(* Logix 5000 project; controller reports 1756-L63 rev 20.11; software revision 20.04; part 33 of 52 *)

        [12].log_data[39].valid := 1, [12].log_data[40].min := 7.5629425, [12].log_data[40].max := 7.590698, [12].log_data[40].total := 27279.617, [12].log_data[40].time := 3600.0, [12].log_data[40].minminute := 8, [12].log_data[40].maxminute := 16, [12].log_data[40].valid := 1, [12].log_data[41].min := 0.03412134, [12].log_data[41].max := 0.0517876, [12].log_data[41].total := 150.64825, [12].log_data[41].time := 3600.0, [12].log_data[41].minminute := 1, [12].log_data[41].maxminute := 24, [12].log_data[41].valid := 1, [12].log_data[42].min := 2.292585, [12].log_data[42].max := 2.2987092, [12].log_data[42].total := 8264.11, [12].log_data[42].time := 3600.0, [12].log_data[42].minminute := 1, [12].log_data[42].maxminute := 32, [12].log_data[42].valid := 1, [12].log_data[43].min := -0.27999878, [12].log_data[43].max := -0.26000214, [12].log_data[43].total := -938.01764, [12].log_data[43].time := 3600.0, [12].log_data[43].valid := 1, [12].log_data[44].min := -0.30000305, [12].log_data[44].max := -0.27999878, [12].log_data[44].total := -1080.081, [12].log_data[44].time := 3600.0, [12].log_data[44].maxminute := 16, [12].log_data[44].valid := 1, [12].log_data[45].time := 3600.0, [12].log_data[45].valid := 1, [12].log_data[46].time := 3600.0, [12].log_data[46].valid := 1, [12].log_data[47].time := 3600.0, [12].log_data[47].valid := 1, [12].log_data[48].min := 6.650855, [12].log_data[48].max := 6.8709764, [12].log_data[48].total := 24089.69, [12].log_data[48].time := 3600.0, [12].log_data[48].minminute := 16, [12].log_data[48].maxminute := 3, [12].log_data[48].valid := 1, [12].log_data[49].min := 7.641001, [12].log_data[49].max := 9.442957, [12].log_data[49].total := 31503.416, [12].log_data[49].time := 3600.0, [12].log_data[49].minminute := 15, [12].log_data[49].maxminute := 59, [12].log_data[49].valid := 1, [12].log_data[50].min := 2.016285, [12].log_data[50].max := 2.093074, [12].log_data[50].total := 7406.019, [12].log_data[50].time := 3600.0, [12].log_data[50].minminute := 59, [12].log_data[50].maxminute := 5, [12].log_data[50].valid := 1,
        [12].log_data[51].time := 3600.0, [12].log_data[51].valid := 1, [12].log_data[52].min := -2.9199982, [12].log_data[52].max := 0.11999512, [12].log_data[52].total := -7511.6816, [12].log_data[52].time := 3600.0, [12].log_data[52].minminute := 12, [12].log_data[52].valid := 1, [12].log_data[53].min := -2.5, [12].log_data[53].max := 0.19999695, [12].log_data[53].total := -7003.9526, [12].log_data[53].time := 3600.0, [12].log_data[53].minminute := 37, [12].log_data[53].maxminute := 15, [12].log_data[53].valid := 1, [12].log_data[54].max := 0.535, [12].log_data[54].total := 1217.1705, [12].log_data[54].time := 3600.0, [12].log_data[54].maxminute := 12, [12].log_data[54].valid := 1, [12].log_data[55].max := 0.51600003, [12].log_data[55].total := 1217.1682, [12].log_data[55].time := 3600.0, [12].log_data[55].minminute := 3, [12].log_data[55].maxminute := 37, [12].log_data[55].valid := 1, [12].log_data[56].min := 0.16024561, [12].log_data[56].max := 0.16063818, [12].log_data[56].total := 577.4149, [12].log_data[56].time := 3600.0, [12].log_data[56].minminute := 10, [12].log_data[56].maxminute := 2, [12].log_data[56].valid := 1, [12].log_data[57].min := 0.31213588, [12].log_data[57].max := 0.3125677, [12].log_data[57].total := 1124.3689, [12].log_data[57].time := 3600.0, [12].log_data[57].minminute := 57, [12].log_data[57].maxminute := 15, [12].log_data[57].valid := 1, [12].log_data[58].time := 3600.0, [12].log_data[58].valid := 1, [12].log_data[59].time := 3600.0, [12].log_data[59].valid := 1, [12].log_data[60].valid := 1, [12].log_data[61].valid := 1, [12].log_data[62].valid := 1, [12].log_data[63].valid := 1, [12].log_data[64].valid := 1, [12].log_data[65].valid := 1, [12].log_data[66].valid := 1, [12].log_data[67].valid := 1, [12].log_data[68].valid := 1, [12].log_data[69].valid := 1, [12].log_data[70].valid := 1, [12].log_data[71].valid := 1, [12].log_data[72].valid := 1, [12].log_data[73].valid := 1, [12].log_data[74].valid := 1, [12].log_data[75].valid := 1,
        [12].log_data[76].valid := 1, [12].log_data[77].valid := 1, [12].log_data[78].valid := 1, [12].log_data[79].valid := 1, [12].log_data[80].valid := 1, [12].log_data[81].valid := 1, [12].log_data[82].valid := 1, [12].log_data[83].valid := 1, [12].log_data[84].valid := 1, [12].log_data[85].valid := 1, [12].log_data[86].valid := 1, [12].log_data[87].valid := 1, [12].log_data[88].valid := 1, [12].log_data[89].valid := 1, [12].log_data[90].valid := 1, [12].log_data[91].valid := 1, [12].log_data[92].valid := 1, [12].log_data[93].valid := 1, [12].log_data[94].valid := 1, [12].log_data[95].valid := 1, [12].log_data[96].valid := 1, [12].log_data[97].valid := 1, [12].log_data[98].valid := 1, [12].log_data[99].valid := 1, [12].log_data[100].valid := 1, [12].log_data[101].valid := 1, [12].log_data[102].valid := 1, [12].log_data[103].valid := 1, [12].log_data[104].valid := 1, [12].log_data[105].valid := 1, [12].log_data[106].valid := 1, [12].log_data[107].valid := 1, [12].log_data[108].valid := 1, [12].log_data[109].valid := 1, [12].log_data[110].valid := 1, [12].log_data[111].valid := 1, [12].log_data[112].valid := 1, [12].log_data[113].valid := 1, [12].log_data[114].valid := 1, [12].log_data[115].valid := 1, [12].log_data[116].valid := 1, [12].log_data[117].valid := 1, [12].log_data[118].valid := 1, [12].log_data[119].valid := 1, [12].log_data[120].valid := 1, [12].log_data[121].valid := 1, [12].log_data[122].valid := 1, [12].log_data[123].valid := 1, [12].log_data[124].valid := 1, [12].time.Year := 2023, [12].time.Month := 1, [12].time.Day := 13, [12].time.Hour := 15, [12].time.Minute := 59, [12].time.Second := 59, [13].log_data[0].min := 1.0, [13].log_data[0].max := 1.0, [13].log_data[0].total := 3600.0, [13].log_data[0].time := 3600.0, [13].log_data[0].valid := 1,
        [13].log_data[1].max := 1.0, [13].log_data[1].total := 530.0, [13].log_data[1].time := 3600.0, [13].log_data[1].maxminute := 20, [13].log_data[1].valid := 1, [13].log_data[2].max := 1.0, [13].log_data[2].total := 526.5, [13].log_data[2].time := 3600.0, [13].log_data[2].maxminute := 20, [13].log_data[2].valid := 1, [13].log_data[3].time := 3600.0, [13].log_data[3].valid := 1, [13].log_data[4].time := 3600.0, [13].log_data[4].valid := 1, [13].log_data[5].max := 1.0, [13].log_data[5].total := 238.5, [13].log_data[5].time := 3600.0, [13].log_data[5].maxminute := 23, [13].log_data[5].valid := 1, [13].log_data[6].time := 3600.0, [13].log_data[6].valid := 1, [13].log_data[7].time := 3600.0, [13].log_data[7].valid := 1, [13].log_data[8].max := 1.0, [13].log_data[8].total := 2819.5, [13].log_data[8].time := 3600.0, [13].log_data[8].minminute := 12, [13].log_data[8].valid := 1, [13].log_data[9].max := 1.0, [13].log_data[9].total := 2816.0, [13].log_data[9].time := 3600.0, [13].log_data[9].minminute := 12, [13].log_data[9].valid := 1, [13].log_data[10].min := 1.0, [13].log_data[10].max := 1.0, [13].log_data[10].total := 3600.0, [13].log_data[10].time := 3600.0, [13].log_data[10].valid := 1, [13].log_data[11].time := 3600.0, [13].log_data[11].valid := 1, [13].log_data[12].min := 1.0, [13].log_data[12].max := 1.0, [13].log_data[12].total := 3600.0, [13].log_data[12].time := 3600.0, [13].log_data[12].valid := 1, [13].log_data[13].min := 1.0, [13].log_data[13].max := 1.0, [13].log_data[13].total := 3600.0, [13].log_data[13].time := 3600.0, [13].log_data[13].valid := 1, [13].log_data[14].time := 3600.0, [13].log_data[14].valid := 1, [13].log_data[15].time := 3600.0, [13].log_data[15].valid := 1, [13].log_data[16].time := 3600.0, [13].log_data[16].valid := 1, [13].log_data[17].min := 1.0, [13].log_data[17].max := 1.0, [13].log_data[17].total := 3600.0, [13].log_data[17].time := 3600.0,
        [13].log_data[17].valid := 1, [13].log_data[18].time := 3600.0, [13].log_data[18].valid := 1, [13].log_data[19].time := 3600.0, [13].log_data[19].valid := 1, [13].log_data[20].time := 3600.0, [13].log_data[20].valid := 1, [13].log_data[21].min := 1.0, [13].log_data[21].max := 1.0, [13].log_data[21].total := 3600.0, [13].log_data[21].time := 3600.0, [13].log_data[21].valid := 1, [13].log_data[22].time := 3600.0, [13].log_data[22].valid := 1, [13].log_data[23].time := 3600.0, [13].log_data[23].valid := 1, [13].log_data[24].time := 3600.0, [13].log_data[24].valid := 1, [13].log_data[25].time := 3600.0, [13].log_data[25].valid := 1, [13].log_data[26].time := 3600.0, [13].log_data[26].valid := 1, [13].log_data[27].time := 3600.0, [13].log_data[27].valid := 1, [13].log_data[28].time := 3600.0, [13].log_data[28].valid := 1, [13].log_data[29].min := 1.0, [13].log_data[29].max := 1.0, [13].log_data[29].total := 3600.0, [13].log_data[29].time := 3600.0, [13].log_data[29].valid := 1, [13].log_data[30].min := 1.0, [13].log_data[30].max := 1.0, [13].log_data[30].total := 3600.0, [13].log_data[30].time := 3600.0, [13].log_data[30].valid := 1, [13].log_data[31].max := 1.0, [13].log_data[31].total := 905.749, [13].log_data[31].time := 3600.0, [13].log_data[31].minminute := 3, [13].log_data[31].valid := 1, [13].log_data[32].max := 1.0, [13].log_data[32].total := 1495.5, [13].log_data[32].time := 3600.0, [13].log_data[32].maxminute := 5, [13].log_data[32].valid := 1, [13].log_data[33].time := 3600.0, [13].log_data[33].valid := 1, [13].log_data[34].time := 3600.0, [13].log_data[34].valid := 1, [13].log_data[35].max := 1.0, [13].log_data[35].total := 1299.749, [13].log_data[35].time := 3600.0, [13].log_data[35].minminute := 7, [13].log_data[35].valid := 1, [13].log_data[36].max := 1.0, [13].log_data[36].total := 1160.247, [13].log_data[36].time := 3600.0, [13].log_data[36].maxminute := 8, [13].log_data[36].valid := 1,
        [13].log_data[37].max := 7.6030836, [13].log_data[37].total := 3481.0479, [13].log_data[37].time := 3600.0, [13].log_data[37].maxminute := 21, [13].log_data[37].valid := 1, [13].log_data[38].time := 3600.0, [13].log_data[38].valid := 1, [13].log_data[39].min := 0.9944707, [13].log_data[39].max := 1.02203, [13].log_data[39].total := 3607.03, [13].log_data[39].time := 3600.0, [13].log_data[39].minminute := 59, [13].log_data[39].maxminute := 27, [13].log_data[39].valid := 1, [13].log_data[40].min := 7.572836, [13].log_data[40].max := 7.5805306, [13].log_data[40].total := 27278.973, [13].log_data[40].time := 3600.0, [13].log_data[40].minminute := 17, [13].log_data[40].maxminute := 49, [13].log_data[40].valid := 1, [13].log_data[41].min := 0.028036376, [13].log_data[41].max := 0.049824707, [13].log_data[41].total := 143.90239, [13].log_data[41].time := 3600.0, [13].log_data[41].minminute := 30, [13].log_data[41].maxminute := 4, [13].log_data[41].valid := 1, [13].log_data[42].min := 2.2929382, [13].log_data[42].max := 2.2984736, [13].log_data[42].total := 8264.059, [13].log_data[42].time := 3600.0, [13].log_data[42].minminute := 7, [13].log_data[42].maxminute := 29, [13].log_data[42].valid := 1, [13].log_data[43].min := -0.27999878, [13].log_data[43].max := -0.26000214, [13].log_data[43].total := -938.47235, [13].log_data[43].time := 3600.0, [13].log_data[43].valid := 1, [13].log_data[44].min := -0.30000305, [13].log_data[44].max := -0.27999878, [13].log_data[44].total := -1080.086, [13].log_data[44].time := 3600.0, [13].log_data[44].maxminute := 46, [13].log_data[44].valid := 1, [13].log_data[45].time := 3600.0, [13].log_data[45].valid := 1, [13].log_data[46].time := 3600.0, [13].log_data[46].valid := 1, [13].log_data[47].time := 3600.0, [13].log_data[47].valid := 1, [13].log_data[48].min := 6.5725355, [13].log_data[48].max := 6.936381, [13].log_data[48].total := 24110.77, [13].log_data[48].time := 3600.0, [13].log_data[48].minminute := 50, [13].log_data[48].maxminute := 29, [13].log_data[48].valid := 1, [13].log_data[49].min := 6.7824225,
        [13].log_data[49].max := 9.446097, [13].log_data[49].total := 29833.777, [13].log_data[49].time := 3600.0, [13].log_data[49].minminute := 48, [13].log_data[49].maxminute := 10, [13].log_data[49].valid := 1, [13].log_data[50].min := 1.9995611, [13].log_data[50].max := 2.1512551, [13].log_data[50].total := 7471.418, [13].log_data[50].time := 3600.0, [13].log_data[50].minminute := 12, [13].log_data[50].maxminute := 25, [13].log_data[50].valid := 1, [13].log_data[51].time := 3600.0, [13].log_data[51].valid := 1, [13].log_data[52].min := -4.220001, [13].log_data[52].max := 0.11999512, [13].log_data[52].total := -6930.1035, [13].log_data[52].time := 3600.0, [13].log_data[52].minminute := 25, [13].log_data[52].maxminute := 3, [13].log_data[52].valid := 1, [13].log_data[53].min := -3.959999, [13].log_data[53].max := 0.19999695, [13].log_data[53].total := -6586.3633, [13].log_data[53].time := 3600.0, [13].log_data[53].minminute := 25, [13].log_data[53].maxminute := 31, [13].log_data[53].valid := 1, [13].log_data[54].max := 0.5435, [13].log_data[54].total := 951.75946, [13].log_data[54].time := 3600.0, [13].log_data[54].minminute := 3, [13].log_data[54].maxminute := 28, [13].log_data[54].valid := 1, [13].log_data[55].max := 0.5385, [13].log_data[55].total := 974.7713, [13].log_data[55].time := 3600.0, [13].log_data[55].minminute := 7, [13].log_data[55].maxminute := 25, [13].log_data[55].valid := 1, [13].log_data[56].min := 0.16020635, [13].log_data[56].max := 0.16059892, [13].log_data[56].total := 577.38025, [13].log_data[56].time := 3600.0, [13].log_data[56].minminute := 53, [13].log_data[56].valid := 1, [13].log_data[57].min := 0.31009445, [13].log_data[57].max := 0.31252846, [13].log_data[57].total := 1123.3262, [13].log_data[57].time := 3600.0, [13].log_data[57].minminute := 59, [13].log_data[57].valid := 1, [13].log_data[58].time := 3600.0, [13].log_data[58].valid := 1, [13].log_data[59].time := 3600.0, [13].log_data[59].valid := 1, [13].log_data[60].valid := 1, [13].log_data[61].valid := 1, [13].log_data[62].valid := 1,
        [13].log_data[63].valid := 1, [13].log_data[64].valid := 1, [13].log_data[65].valid := 1, [13].log_data[66].valid := 1, [13].log_data[67].valid := 1, [13].log_data[68].valid := 1, [13].log_data[69].valid := 1, [13].log_data[70].valid := 1, [13].log_data[71].valid := 1, [13].log_data[72].valid := 1, [13].log_data[73].valid := 1, [13].log_data[74].valid := 1, [13].log_data[75].valid := 1, [13].log_data[76].valid := 1, [13].log_data[77].valid := 1, [13].log_data[78].valid := 1, [13].log_data[79].valid := 1, [13].log_data[80].valid := 1, [13].log_data[81].valid := 1, [13].log_data[82].valid := 1, [13].log_data[83].valid := 1, [13].log_data[84].valid := 1, [13].log_data[85].valid := 1, [13].log_data[86].valid := 1, [13].log_data[87].valid := 1, [13].log_data[88].valid := 1, [13].log_data[89].valid := 1, [13].log_data[90].valid := 1, [13].log_data[91].valid := 1, [13].log_data[92].valid := 1, [13].log_data[93].valid := 1, [13].log_data[94].valid := 1, [13].log_data[95].valid := 1, [13].log_data[96].valid := 1, [13].log_data[97].valid := 1, [13].log_data[98].valid := 1, [13].log_data[99].valid := 1, [13].log_data[100].valid := 1, [13].log_data[101].valid := 1, [13].log_data[102].valid := 1, [13].log_data[103].valid := 1, [13].log_data[104].valid := 1, [13].log_data[105].valid := 1, [13].log_data[106].valid := 1, [13].log_data[107].valid := 1, [13].log_data[108].valid := 1, [13].log_data[109].valid := 1, [13].log_data[110].valid := 1, [13].log_data[111].valid := 1, [13].log_data[112].valid := 1, [13].log_data[113].valid := 1, [13].log_data[114].valid := 1, [13].log_data[115].valid := 1, [13].log_data[116].valid := 1, [13].log_data[117].valid := 1, [13].log_data[118].valid := 1, [13].log_data[119].valid := 1, [13].log_data[120].valid := 1, [13].log_data[121].valid := 1, [13].log_data[122].valid := 1,
        [13].log_data[123].valid := 1, [13].log_data[124].valid := 1, [13].time.Year := 2023, [13].time.Month := 1, [13].time.Day := 13, [13].time.Hour := 16, [13].time.Minute := 59, [13].time.Second := 59, [14].log_data[0].min := 1.0, [14].log_data[0].max := 1.0, [14].log_data[0].total := 3600.0, [14].log_data[0].time := 3600.0, [14].log_data[0].valid := 1, [14].log_data[1].time := 3600.0, [14].log_data[1].valid := 1, [14].log_data[2].time := 3600.0, [14].log_data[2].valid := 1, [14].log_data[3].time := 3600.0, [14].log_data[3].valid := 1, [14].log_data[4].time := 3600.0, [14].log_data[4].valid := 1, [14].log_data[5].time := 3600.0, [14].log_data[5].valid := 1, [14].log_data[6].time := 3600.0, [14].log_data[6].valid := 1, [14].log_data[7].time := 3600.0, [14].log_data[7].valid := 1, [14].log_data[8].max := 1.0, [14].log_data[8].total := 3099.251, [14].log_data[8].time := 3600.0, [14].log_data[8].minminute := 51, [14].log_data[8].valid := 1, [14].log_data[9].max := 1.0, [14].log_data[9].total := 3099.251, [14].log_data[9].time := 3600.0, [14].log_data[9].minminute := 51, [14].log_data[9].valid := 1, [14].log_data[10].min := 1.0, [14].log_data[10].max := 1.0, [14].log_data[10].total := 3600.0, [14].log_data[10].time := 3600.0, [14].log_data[10].valid := 1, [14].log_data[11].time := 3600.0, [14].log_data[11].valid := 1, [14].log_data[12].min := 1.0, [14].log_data[12].max := 1.0, [14].log_data[12].total := 3600.0, [14].log_data[12].time := 3600.0, [14].log_data[12].valid := 1, [14].log_data[13].min := 1.0, [14].log_data[13].max := 1.0, [14].log_data[13].total := 3600.0, [14].log_data[13].time := 3600.0, [14].log_data[13].valid := 1, [14].log_data[14].time := 3600.0, [14].log_data[14].valid := 1, [14].log_data[15].time := 3600.0, [14].log_data[15].valid := 1, [14].log_data[16].time := 3600.0, [14].log_data[16].valid := 1,
        [14].log_data[17].min := 1.0, [14].log_data[17].max := 1.0, [14].log_data[17].total := 3600.0, [14].log_data[17].time := 3600.0, [14].log_data[17].valid := 1, [14].log_data[18].time := 3600.0, [14].log_data[18].valid := 1, [14].log_data[19].time := 3600.0, [14].log_data[19].valid := 1, [14].log_data[20].time := 3600.0, [14].log_data[20].valid := 1, [14].log_data[21].min := 1.0, [14].log_data[21].max := 1.0, [14].log_data[21].total := 3600.0, [14].log_data[21].time := 3600.0, [14].log_data[21].valid := 1, [14].log_data[22].time := 3600.0, [14].log_data[22].valid := 1, [14].log_data[23].time := 3600.0, [14].log_data[23].valid := 1, [14].log_data[24].time := 3600.0, [14].log_data[24].valid := 1, [14].log_data[25].time := 3600.0, [14].log_data[25].valid := 1, [14].log_data[26].time := 3600.0, [14].log_data[26].valid := 1, [14].log_data[27].time := 3600.0, [14].log_data[27].valid := 1, [14].log_data[28].time := 3600.0, [14].log_data[28].valid := 1, [14].log_data[29].min := 1.0, [14].log_data[29].max := 1.0, [14].log_data[29].total := 3600.0, [14].log_data[29].time := 3600.0, [14].log_data[29].valid := 1, [14].log_data[30].min := 1.0, [14].log_data[30].max := 1.0, [14].log_data[30].total := 3600.0, [14].log_data[30].time := 3600.0, [14].log_data[30].valid := 1, [14].log_data[31].max := 1.0, [14].log_data[31].total := 1629.998, [14].log_data[31].time := 3600.0, [14].log_data[31].valid := 1, [14].log_data[32].max := 1.0, [14].log_data[32].total := 1086.498, [14].log_data[32].time := 3600.0, [14].log_data[32].maxminute := 10, [14].log_data[32].valid := 1, [14].log_data[33].time := 3600.0, [14].log_data[33].valid := 1, [14].log_data[34].time := 3600.0, [14].log_data[34].valid := 1, [14].log_data[35].max := 1.0, [14].log_data[35].total := 1437.7471, [14].log_data[35].time := 3600.0, [14].log_data[35].maxminute := 3, [14].log_data[35].valid := 1, [14].log_data[36].max := 1.0, [14].log_data[36].total := 1223.998,
        [14].log_data[36].time := 3600.0, [14].log_data[36].minminute := 2, [14].log_data[36].valid := 1, [14].log_data[37].time := 3600.0, [14].log_data[37].valid := 1, [14].log_data[38].time := 3600.0, [14].log_data[38].valid := 1, [14].log_data[39].min := 0.9935285, [14].log_data[39].max := 1.005306, [14].log_data[39].total := 3600.2817, [14].log_data[39].time := 3600.0, [14].log_data[39].minminute := 35, [14].log_data[39].maxminute := 25, [14].log_data[39].valid := 1, [14].log_data[40].min := 7.5717363, [14].log_data[40].max := 7.5838275, [14].log_data[40].total := 27280.795, [14].log_data[40].time := 3600.0, [14].log_data[40].minminute := 19, [14].log_data[40].maxminute := 28, [14].log_data[40].valid := 1, [14].log_data[41].min := 0.042365476, [14].log_data[41].max := 0.061994627, [14].log_data[41].total := 193.76056, [14].log_data[41].time := 3600.0, [14].log_data[41].minminute := 59, [14].log_data[41].maxminute := 10, [14].log_data[41].valid := 1, [14].log_data[42].min := 2.2928205, [14].log_data[42].max := 2.2983558, [14].log_data[42].total := 8264.156, [14].log_data[42].time := 3600.0, [14].log_data[42].minminute := 9, [14].log_data[42].maxminute := 33, [14].log_data[42].valid := 1, [14].log_data[43].min := -0.27999878, [14].log_data[43].max := -0.26000214, [14].log_data[43].total := -936.9969, [14].log_data[43].time := 3600.0, [14].log_data[43].valid := 1, [14].log_data[44].min := -0.30000305, [14].log_data[44].max := -0.27999878, [14].log_data[44].total := -1079.9506, [14].log_data[44].time := 3600.0, [14].log_data[44].maxminute := 2, [14].log_data[44].valid := 1, [14].log_data[45].time := 3600.0, [14].log_data[45].valid := 1, [14].log_data[46].time := 3600.0, [14].log_data[46].valid := 1, [14].log_data[47].time := 3600.0, [14].log_data[47].valid := 1, [14].log_data[48].min := 6.734946, [14].log_data[48].max := 6.7967777, [14].log_data[48].total := 24332.396, [14].log_data[48].time := 3600.0, [14].log_data[48].maxminute := 5, [14].log_data[48].valid := 1, [14].log_data[49].min := 7.6767263, [14].log_data[49].max := 9.449238,
        [14].log_data[49].total := 32822.707, [14].log_data[49].time := 3600.0, [14].log_data[49].maxminute := 51, [14].log_data[49].valid := 1, [14].log_data[50].min := 1.9990901, [14].log_data[50].max := 2.0975497, [14].log_data[50].total := 7358.2993, [14].log_data[50].time := 3600.0, [14].log_data[50].minminute := 51, [14].log_data[50].maxminute := 59, [14].log_data[50].valid := 1, [14].log_data[51].time := 3600.0, [14].log_data[51].valid := 1, [14].log_data[52].min := -2.9400024, [14].log_data[52].max := 0.11999512, [14].log_data[52].total := -7247.679, [14].log_data[52].time := 3600.0, [14].log_data[52].minminute := 11, [14].log_data[52].valid := 1, [14].log_data[53].min := -2.6200027, [14].log_data[53].max := 0.17999268, [14].log_data[53].total := -6591.616, [14].log_data[53].time := 3600.0, [14].log_data[53].minminute := 3, [14].log_data[53].maxminute := 13, [14].log_data[53].valid := 1, [14].log_data[54].max := 0.5385, [14].log_data[54].total := 1077.6411, [14].log_data[54].time := 3600.0, [14].log_data[54].maxminute := 32, [14].log_data[54].valid := 1, [14].log_data[55].max := 0.532, [14].log_data[55].total := 1055.9913, [14].log_data[55].time := 3600.0, [14].log_data[55].minminute := 2, [14].log_data[55].maxminute := 14, [14].log_data[55].valid := 1, [14].log_data[56].min := 0.16024561, [14].log_data[56].max := 0.16063818, [14].log_data[56].total := 577.48267, [14].log_data[56].time := 3600.0, [14].log_data[56].minminute := 18, [14].log_data[56].maxminute := 20, [14].log_data[56].valid := 1, [14].log_data[57].min := 0.30997667, [14].log_data[57].max := 0.31040853, [14].log_data[57].total := 1116.629, [14].log_data[57].time := 3600.0, [14].log_data[57].minminute := 6, [14].log_data[57].maxminute := 38, [14].log_data[57].valid := 1, [14].log_data[58].time := 3600.0, [14].log_data[58].valid := 1, [14].log_data[59].time := 3600.0, [14].log_data[59].valid := 1, [14].log_data[60].valid := 1, [14].log_data[61].valid := 1, [14].log_data[62].valid := 1, [14].log_data[63].valid := 1, [14].log_data[64].valid := 1,
        [14].log_data[65].valid := 1, [14].log_data[66].valid := 1, [14].log_data[67].valid := 1, [14].log_data[68].valid := 1, [14].log_data[69].valid := 1, [14].log_data[70].valid := 1, [14].log_data[71].valid := 1, [14].log_data[72].valid := 1, [14].log_data[73].valid := 1, [14].log_data[74].valid := 1, [14].log_data[75].valid := 1, [14].log_data[76].valid := 1, [14].log_data[77].valid := 1, [14].log_data[78].valid := 1, [14].log_data[79].valid := 1, [14].log_data[80].valid := 1, [14].log_data[81].valid := 1, [14].log_data[82].valid := 1, [14].log_data[83].valid := 1, [14].log_data[84].valid := 1, [14].log_data[85].valid := 1, [14].log_data[86].valid := 1, [14].log_data[87].valid := 1, [14].log_data[88].valid := 1, [14].log_data[89].valid := 1, [14].log_data[90].valid := 1, [14].log_data[91].valid := 1, [14].log_data[92].valid := 1, [14].log_data[93].valid := 1, [14].log_data[94].valid := 1, [14].log_data[95].valid := 1, [14].log_data[96].valid := 1, [14].log_data[97].valid := 1, [14].log_data[98].valid := 1, [14].log_data[99].valid := 1, [14].log_data[100].valid := 1, [14].log_data[101].valid := 1, [14].log_data[102].valid := 1, [14].log_data[103].valid := 1, [14].log_data[104].valid := 1, [14].log_data[105].valid := 1, [14].log_data[106].valid := 1, [14].log_data[107].valid := 1, [14].log_data[108].valid := 1, [14].log_data[109].valid := 1, [14].log_data[110].valid := 1, [14].log_data[111].valid := 1, [14].log_data[112].valid := 1, [14].log_data[113].valid := 1, [14].log_data[114].valid := 1, [14].log_data[115].valid := 1, [14].log_data[116].valid := 1, [14].log_data[117].valid := 1, [14].log_data[118].valid := 1, [14].log_data[119].valid := 1, [14].log_data[120].valid := 1, [14].log_data[121].valid := 1, [14].log_data[122].valid := 1, [14].log_data[123].valid := 1, [14].log_data[124].valid := 1,
        [14].time.Year := 2023, [14].time.Month := 1, [14].time.Day := 13, [14].time.Hour := 17, [14].time.Minute := 59, [14].time.Second := 59, [15].log_data[0].min := 1.0, [15].log_data[0].max := 1.0, [15].log_data[0].total := 3600.0, [15].log_data[0].time := 3600.0, [15].log_data[0].valid := 1, [15].log_data[1].max := 1.0, [15].log_data[1].total := 572.0, [15].log_data[1].time := 3600.0, [15].log_data[1].maxminute := 18, [15].log_data[1].valid := 1, [15].log_data[2].max := 1.0, [15].log_data[2].total := 568.5, [15].log_data[2].time := 3600.0, [15].log_data[2].maxminute := 18, [15].log_data[2].valid := 1, [15].log_data[3].time := 3600.0, [15].log_data[3].valid := 1, [15].log_data[4].time := 3600.0, [15].log_data[4].valid := 1, [15].log_data[5].max := 1.0, [15].log_data[5].total := 230.0, [15].log_data[5].time := 3600.0, [15].log_data[5].maxminute := 21, [15].log_data[5].valid := 1, [15].log_data[6].time := 3600.0, [15].log_data[6].valid := 1, [15].log_data[7].time := 3600.0, [15].log_data[7].valid := 1, [15].log_data[8].max := 1.0, [15].log_data[8].total := 2202.249, [15].log_data[8].time := 3600.0, [15].log_data[8].maxminute := 23, [15].log_data[8].valid := 1, [15].log_data[9].max := 1.0, [15].log_data[9].total := 2198.749, [15].log_data[9].time := 3600.0, [15].log_data[9].maxminute := 23, [15].log_data[9].valid := 1, [15].log_data[10].min := 1.0, [15].log_data[10].max := 1.0, [15].log_data[10].total := 3600.0, [15].log_data[10].time := 3600.0, [15].log_data[10].valid := 1, [15].log_data[11].time := 3600.0, [15].log_data[11].valid := 1, [15].log_data[12].min := 1.0, [15].log_data[12].max := 1.0, [15].log_data[12].total := 3600.0, [15].log_data[12].time := 3600.0, [15].log_data[12].valid := 1, [15].log_data[13].min := 1.0, [15].log_data[13].max := 1.0, [15].log_data[13].total := 3600.0, [15].log_data[13].time := 3600.0,
        [15].log_data[13].valid := 1, [15].log_data[14].time := 3600.0, [15].log_data[14].valid := 1, [15].log_data[15].time := 3600.0, [15].log_data[15].valid := 1, [15].log_data[16].time := 3600.0, [15].log_data[16].valid := 1, [15].log_data[17].min := 1.0, [15].log_data[17].max := 1.0, [15].log_data[17].total := 3600.0, [15].log_data[17].time := 3600.0, [15].log_data[17].valid := 1, [15].log_data[18].time := 3600.0, [15].log_data[18].valid := 1, [15].log_data[19].time := 3600.0, [15].log_data[19].valid := 1, [15].log_data[20].time := 3600.0, [15].log_data[20].valid := 1, [15].log_data[21].min := 1.0, [15].log_data[21].max := 1.0, [15].log_data[21].total := 3600.0, [15].log_data[21].time := 3600.0, [15].log_data[21].valid := 1, [15].log_data[22].time := 3600.0, [15].log_data[22].valid := 1, [15].log_data[23].time := 3600.0, [15].log_data[23].valid := 1, [15].log_data[24].time := 3600.0, [15].log_data[24].valid := 1, [15].log_data[25].time := 3600.0, [15].log_data[25].valid := 1, [15].log_data[26].time := 3600.0, [15].log_data[26].valid := 1, [15].log_data[27].time := 3600.0, [15].log_data[27].valid := 1, [15].log_data[28].time := 3600.0, [15].log_data[28].valid := 1, [15].log_data[29].min := 1.0, [15].log_data[29].max := 1.0, [15].log_data[29].total := 3600.0, [15].log_data[29].time := 3600.0, [15].log_data[29].valid := 1, [15].log_data[30].min := 1.0, [15].log_data[30].max := 1.0, [15].log_data[30].total := 3600.0, [15].log_data[30].time := 3600.0, [15].log_data[30].valid := 1, [15].log_data[31].max := 1.0, [15].log_data[31].total := 843.99805, [15].log_data[31].time := 3600.0, [15].log_data[31].maxminute := 33, [15].log_data[31].valid := 1, [15].log_data[32].max := 1.0, [15].log_data[32].total := 1086.498, [15].log_data[32].time := 3600.0, [15].log_data[32].maxminute := 23, [15].log_data[32].valid := 1, [15].log_data[33].time := 3600.0, [15].log_data[33].valid := 1, [15].log_data[34].time := 3600.0,
        [15].log_data[34].valid := 1, [15].log_data[35].max := 1.0, [15].log_data[35].total := 1086.498, [15].log_data[35].time := 3600.0, [15].log_data[35].maxminute := 28, [15].log_data[35].valid := 1, [15].log_data[36].max := 1.0, [15].log_data[36].total := 752.247, [15].log_data[36].time := 3600.0, [15].log_data[36].maxminute := 23, [15].log_data[36].valid := 1, [15].log_data[37].max := 7.0664234, [15].log_data[37].total := 3536.743, [15].log_data[37].time := 3600.0, [15].log_data[37].maxminute := 22, [15].log_data[37].valid := 1, [15].log_data[38].time := 3600.0, [15].log_data[38].valid := 1, [15].log_data[39].min := 0.99305737, [15].log_data[39].max := 1.0216767, [15].log_data[39].total := 3608.93, [15].log_data[39].time := 3600.0, [15].log_data[39].minminute := 17, [15].log_data[39].maxminute := 21, [15].log_data[39].valid := 1, [15].log_data[40].min := 7.546179, [15].log_data[40].max := 7.593721, [15].log_data[40].total := 27269.342, [15].log_data[40].time := 3600.0, [15].log_data[40].minminute := 25, [15].log_data[40].maxminute := 18, [15].log_data[40].valid := 1, [15].log_data[41].min := 0.03412134, [15].log_data[41].max := 0.047469236, [15].log_data[41].total := 149.91223, [15].log_data[41].time := 3600.0, [15].log_data[41].minminute := 21, [15].log_data[41].maxminute := 57, [15].log_data[41].valid := 1, [15].log_data[42].min := 2.2927027, [15].log_data[42].max := 2.2978847, [15].log_data[42].total := 8263.865, [15].log_data[42].time := 3600.0, [15].log_data[42].minminute := 29, [15].log_data[42].maxminute := 44, [15].log_data[42].valid := 1, [15].log_data[43].min := -0.27999878, [15].log_data[43].max := -0.26000214, [15].log_data[43].total := -942.1734, [15].log_data[43].time := 3600.0, [15].log_data[43].valid := 1, [15].log_data[44].min := -0.30000305, [15].log_data[44].max := -0.27999878, [15].log_data[44].total := -1080.056, [15].log_data[44].time := 3600.0, [15].log_data[44].maxminute := 3, [15].log_data[44].valid := 1, [15].log_data[45].time := 3600.0, [15].log_data[45].valid := 1, [15].log_data[46].time := 3600.0,
        [15].log_data[46].valid := 1, [15].log_data[47].time := 3600.0, [15].log_data[47].valid := 1, [15].log_data[48].min := 6.58655, [15].log_data[48].max := 6.982273, [15].log_data[48].total := 24215.87, [15].log_data[48].time := 3600.0, [15].log_data[48].minminute := 51, [15].log_data[48].maxminute := 28, [15].log_data[48].valid := 1, [15].log_data[49].min := 6.874287, [15].log_data[49].max := 9.449238, [15].log_data[49].total := 29922.498, [15].log_data[49].time := 3600.0, [15].log_data[49].minminute := 46, [15].log_data[49].maxminute := 5, [15].log_data[49].valid := 1, [15].log_data[50].min := 2.0588017, [15].log_data[50].max := 2.1505485, [15].log_data[50].total := 7536.4956, [15].log_data[50].time := 3600.0, [15].log_data[50].minminute := 25, [15].log_data[50].maxminute := 23, [15].log_data[50].valid := 1, [15].log_data[51].time := 3600.0, [15].log_data[51].valid := 1, [15].log_data[52].min := -4.1800003, [15].log_data[52].max := 0.11999512, [15].log_data[52].total := -6905.693, [15].log_data[52].time := 3600.0, [15].log_data[52].minminute := 23, [15].log_data[52].maxminute := 32, [15].log_data[52].valid := 1, [15].log_data[53].min := -3.9799957, [15].log_data[53].max := 0.17999268, [15].log_data[53].total := -6247.879, [15].log_data[53].time := 3600.0, [15].log_data[53].minminute := 23, [15].log_data[53].maxminute := 48, [15].log_data[53].valid := 1, [15].log_data[54].max := 0.552, [15].log_data[54].total := 764.73987, [15].log_data[54].time := 3600.0, [15].log_data[54].maxminute := 55, [15].log_data[54].valid := 1, [15].log_data[55].max := 0.533, [15].log_data[55].total := 726.16895, [15].log_data[55].time := 3600.0, [15].log_data[55].maxminute := 49, [15].log_data[55].valid := 1, [15].log_data[56].min := 0.16020635, [15].log_data[56].max := 0.16063818, [15].log_data[56].total := 577.4228, [15].log_data[56].time := 3600.0, [15].log_data[56].minminute := 54, [15].log_data[56].valid := 1, [15].log_data[57].min := 0.30832782, [15].log_data[57].max := 0.31040853, [15].log_data[57].total := 1115.9126, [15].log_data[57].time := 3600.0,
        [15].log_data[57].minminute := 58, [15].log_data[57].maxminute := 11, [15].log_data[57].valid := 1, [15].log_data[58].time := 3600.0, [15].log_data[58].valid := 1, [15].log_data[59].time := 3600.0, [15].log_data[59].valid := 1, [15].log_data[60].valid := 1, [15].log_data[61].valid := 1, [15].log_data[62].valid := 1, [15].log_data[63].valid := 1, [15].log_data[64].valid := 1, [15].log_data[65].valid := 1, [15].log_data[66].valid := 1, [15].log_data[67].valid := 1, [15].log_data[68].valid := 1, [15].log_data[69].valid := 1, [15].log_data[70].valid := 1, [15].log_data[71].valid := 1, [15].log_data[72].valid := 1, [15].log_data[73].valid := 1, [15].log_data[74].valid := 1, [15].log_data[75].valid := 1, [15].log_data[76].valid := 1, [15].log_data[77].valid := 1, [15].log_data[78].valid := 1, [15].log_data[79].valid := 1, [15].log_data[80].valid := 1, [15].log_data[81].valid := 1, [15].log_data[82].valid := 1, [15].log_data[83].valid := 1, [15].log_data[84].valid := 1, [15].log_data[85].valid := 1, [15].log_data[86].valid := 1, [15].log_data[87].valid := 1, [15].log_data[88].valid := 1, [15].log_data[89].valid := 1, [15].log_data[90].valid := 1, [15].log_data[91].valid := 1, [15].log_data[92].valid := 1, [15].log_data[93].valid := 1, [15].log_data[94].valid := 1, [15].log_data[95].valid := 1, [15].log_data[96].valid := 1, [15].log_data[97].valid := 1, [15].log_data[98].valid := 1, [15].log_data[99].valid := 1, [15].log_data[100].valid := 1, [15].log_data[101].valid := 1, [15].log_data[102].valid := 1, [15].log_data[103].valid := 1, [15].log_data[104].valid := 1, [15].log_data[105].valid := 1, [15].log_data[106].valid := 1, [15].log_data[107].valid := 1, [15].log_data[108].valid := 1, [15].log_data[109].valid := 1, [15].log_data[110].valid := 1, [15].log_data[111].valid := 1, [15].log_data[112].valid := 1,
        [15].log_data[113].valid := 1, [15].log_data[114].valid := 1, [15].log_data[115].valid := 1, [15].log_data[116].valid := 1, [15].log_data[117].valid := 1, [15].log_data[118].valid := 1, [15].log_data[119].valid := 1, [15].log_data[120].valid := 1, [15].log_data[121].valid := 1, [15].log_data[122].valid := 1, [15].log_data[123].valid := 1, [15].log_data[124].valid := 1, [15].time.Year := 2023, [15].time.Month := 1, [15].time.Day := 13, [15].time.Hour := 18, [15].time.Minute := 59, [15].time.Second := 59, [16].log_data[0].min := 1.0, [16].log_data[0].max := 1.0, [16].log_data[0].total := 3600.0, [16].log_data[0].time := 3600.0, [16].log_data[0].valid := 1, [16].log_data[1].max := 1.0, [16].log_data[1].total := 2.249, [16].log_data[1].time := 3600.0, [16].log_data[1].maxminute := 59, [16].log_data[1].valid := 1, [16].log_data[2].time := 3600.0, [16].log_data[2].valid := 1, [16].log_data[3].time := 3600.0, [16].log_data[3].valid := 1, [16].log_data[4].time := 3600.0, [16].log_data[4].valid := 1, [16].log_data[5].time := 3600.0, [16].log_data[5].valid := 1, [16].log_data[6].time := 3600.0, [16].log_data[6].valid := 1, [16].log_data[7].time := 3600.0, [16].log_data[7].valid := 1, [16].log_data[8].max := 1.0, [16].log_data[8].total := 2742.251, [16].log_data[8].time := 3600.0, [16].log_data[8].minminute := 45, [16].log_data[8].valid := 1, [16].log_data[9].max := 1.0, [16].log_data[9].total := 2742.251, [16].log_data[9].time := 3600.0, [16].log_data[9].minminute := 45, [16].log_data[9].valid := 1, [16].log_data[10].min := 1.0, [16].log_data[10].max := 1.0, [16].log_data[10].total := 3600.0, [16].log_data[10].time := 3600.0, [16].log_data[10].valid := 1, [16].log_data[11].time := 3600.0, [16].log_data[11].valid := 1, [16].log_data[12].min := 1.0, [16].log_data[12].max := 1.0, [16].log_data[12].total := 3600.0,
        [16].log_data[12].time := 3600.0, [16].log_data[12].valid := 1, [16].log_data[13].min := 1.0, [16].log_data[13].max := 1.0, [16].log_data[13].total := 3600.0, [16].log_data[13].time := 3600.0, [16].log_data[13].valid := 1, [16].log_data[14].time := 3600.0, [16].log_data[14].valid := 1, [16].log_data[15].time := 3600.0, [16].log_data[15].valid := 1, [16].log_data[16].time := 3600.0, [16].log_data[16].valid := 1, [16].log_data[17].min := 1.0, [16].log_data[17].max := 1.0, [16].log_data[17].total := 3600.0, [16].log_data[17].time := 3600.0, [16].log_data[17].valid := 1, [16].log_data[18].time := 3600.0, [16].log_data[18].valid := 1, [16].log_data[19].time := 3600.0, [16].log_data[19].valid := 1, [16].log_data[20].time := 3600.0, [16].log_data[20].valid := 1, [16].log_data[21].min := 1.0, [16].log_data[21].max := 1.0, [16].log_data[21].total := 3600.0, [16].log_data[21].time := 3600.0, [16].log_data[21].valid := 1, [16].log_data[22].time := 3600.0, [16].log_data[22].valid := 1, [16].log_data[23].time := 3600.0, [16].log_data[23].valid := 1, [16].log_data[24].time := 3600.0, [16].log_data[24].valid := 1, [16].log_data[25].time := 3600.0, [16].log_data[25].valid := 1, [16].log_data[26].time := 3600.0, [16].log_data[26].valid := 1, [16].log_data[27].time := 3600.0, [16].log_data[27].valid := 1, [16].log_data[28].time := 3600.0, [16].log_data[28].valid := 1, [16].log_data[29].min := 1.0, [16].log_data[29].max := 1.0, [16].log_data[29].total := 3600.0, [16].log_data[29].time := 3600.0, [16].log_data[29].valid := 1, [16].log_data[30].min := 1.0, [16].log_data[30].max := 1.0, [16].log_data[30].total := 3600.0, [16].log_data[30].time := 3600.0, [16].log_data[30].valid := 1, [16].log_data[31].max := 1.0, [16].log_data[31].total := 1306.5, [16].log_data[31].time := 3600.0, [16].log_data[31].minminute := 4, [16].log_data[31].valid := 1, [16].log_data[32].max := 1.0, [16].log_data[32].total := 1086.498,
        [16].log_data[32].time := 3600.0, [16].log_data[32].maxminute := 5, [16].log_data[32].valid := 1, [16].log_data[33].time := 3600.0, [16].log_data[33].valid := 1, [16].log_data[34].time := 3600.0, [16].log_data[34].valid := 1, [16].log_data[35].max := 1.0, [16].log_data[35].total := 1086.498, [16].log_data[35].time := 3600.0, [16].log_data[35].maxminute := 10, [16].log_data[35].valid := 1, [16].log_data[36].max := 1.0, [16].log_data[36].total := 1306.498, [16].log_data[36].time := 3600.0, [16].log_data[36].minminute := 8, [16].log_data[36].valid := 1, [16].log_data[37].max := 4.9178176, [16].log_data[37].total := 12.625217, [16].log_data[37].time := 3600.0, [16].log_data[37].maxminute := 59, [16].log_data[37].valid := 1, [16].log_data[38].time := 3600.0, [16].log_data[38].valid := 1, [16].log_data[39].min := 0.9947063, [16].log_data[39].max := 1.0074259, [16].log_data[39].total := 3607.745, [16].log_data[39].time := 3600.0, [16].log_data[39].minminute := 12, [16].log_data[39].maxminute := 57, [16].log_data[39].valid := 1, [16].log_data[40].min := 7.560194, [16].log_data[40].max := 7.592072, [16].log_data[40].total := 27280.066, [16].log_data[40].time := 3600.0, [16].log_data[40].minminute := 1, [16].log_data[40].maxminute := 4, [16].log_data[40].valid := 1, [16].log_data[41].min := 0.041187745, [16].log_data[41].max := 0.06906128, [16].log_data[41].total := 194.73439, [16].log_data[41].time := 3600.0, [16].log_data[41].minminute := 11, [16].log_data[41].maxminute := 50, [16].log_data[41].valid := 1, [16].log_data[42].min := 2.2929382, [16].log_data[42].max := 2.2985914, [16].log_data[42].total := 8263.699, [16].log_data[42].time := 3600.0, [16].log_data[42].minminute := 18, [16].log_data[42].maxminute := 38, [16].log_data[42].valid := 1, [16].log_data[43].min := -0.27999878, [16].log_data[43].max := -0.26000214, [16].log_data[43].total := -976.6778, [16].log_data[43].time := 3600.0, [16].log_data[43].valid := 1, [16].log_data[44].min := -0.3199997, [16].log_data[44].max := -0.30000305, [16].log_data[44].total := -1080.0961,
        [16].log_data[44].time := 3600.0, [16].log_data[44].minminute := 19, [16].log_data[44].valid := 1, [16].log_data[45].time := 3600.0, [16].log_data[45].valid := 1, [16].log_data[46].time := 3600.0, [16].log_data[46].valid := 1, [16].log_data[47].time := 3600.0, [16].log_data[47].valid := 1, [16].log_data[48].min := 6.733847, [16].log_data[48].max := 6.7984266, [16].log_data[48].total := 24349.666, [16].log_data[48].time := 3600.0, [16].log_data[48].maxminute := 6, [16].log_data[48].valid := 1, [16].log_data[49].min := 8.092472, [16].log_data[49].max := 9.484767, [16].log_data[49].total := 33248.035, [16].log_data[49].time := 3600.0, [16].log_data[49].maxminute := 46, [16].log_data[49].valid := 1, [16].log_data[50].min := 1.9993255, [16].log_data[50].max := 2.1032028, [16].log_data[50].total := 7369.665, [16].log_data[50].time := 3600.0, [16].log_data[50].minminute := 45, [16].log_data[50].maxminute := 59, [16].log_data[50].valid := 1, [16].log_data[51].time := 3600.0, [16].log_data[51].valid := 1, [16].log_data[52].min := -2.8199997, [16].log_data[52].max := 0.11999512, [16].log_data[52].total := -6927.4365, [16].log_data[52].time := 3600.0, [16].log_data[52].minminute := 26, [16].log_data[52].maxminute := 4, [16].log_data[52].valid := 1, [16].log_data[53].min := -2.4600067, [16].log_data[53].max := 0.2599945, [16].log_data[53].total := -6436.3936, [16].log_data[53].time := 3600.0, [16].log_data[53].minminute := 38, [16].log_data[53].maxminute := 20, [16].log_data[53].valid := 1, [16].log_data[54].max := 0.537, [16].log_data[54].total := 950.3685, [16].log_data[54].time := 3600.0, [16].log_data[54].minminute := 4, [16].log_data[54].maxminute := 26, [16].log_data[54].valid := 1, [16].log_data[55].max := 0.50450003, [16].log_data[55].total := 949.557, [16].log_data[55].time := 3600.0, [16].log_data[55].minminute := 8, [16].log_data[55].maxminute := 31, [16].log_data[55].valid := 1, [16].log_data[56].min := 0.16020635, [16].log_data[56].max := 0.16063818, [16].log_data[56].total := 577.4151, [16].log_data[56].time := 3600.0,
        [16].log_data[56].minminute := 57, [16].log_data[56].maxminute := 48, [16].log_data[56].valid := 1, [16].log_data[57].min := 0.30824932, [16].log_data[57].max := 0.30864188, [16].log_data[57].total := 1110.2234, [16].log_data[57].time := 3600.0, [16].log_data[57].minminute := 31, [16].log_data[57].valid := 1, [16].log_data[58].time := 3600.0, [16].log_data[58].valid := 1, [16].log_data[59].time := 3600.0, [16].log_data[59].valid := 1, [16].log_data[60].valid := 1, [16].log_data[61].valid := 1, [16].log_data[62].valid := 1, [16].log_data[63].valid := 1, [16].log_data[64].valid := 1, [16].log_data[65].valid := 1, [16].log_data[66].valid := 1, [16].log_data[67].valid := 1, [16].log_data[68].valid := 1, [16].log_data[69].valid := 1, [16].log_data[70].valid := 1, [16].log_data[71].valid := 1, [16].log_data[72].valid := 1, [16].log_data[73].valid := 1, [16].log_data[74].valid := 1, [16].log_data[75].valid := 1, [16].log_data[76].valid := 1, [16].log_data[77].valid := 1, [16].log_data[78].valid := 1, [16].log_data[79].valid := 1, [16].log_data[80].valid := 1, [16].log_data[81].valid := 1, [16].log_data[82].valid := 1, [16].log_data[83].valid := 1, [16].log_data[84].valid := 1, [16].log_data[85].valid := 1, [16].log_data[86].valid := 1, [16].log_data[87].valid := 1, [16].log_data[88].valid := 1, [16].log_data[89].valid := 1, [16].log_data[90].valid := 1, [16].log_data[91].valid := 1, [16].log_data[92].valid := 1, [16].log_data[93].valid := 1, [16].log_data[94].valid := 1, [16].log_data[95].valid := 1, [16].log_data[96].valid := 1, [16].log_data[97].valid := 1, [16].log_data[98].valid := 1, [16].log_data[99].valid := 1, [16].log_data[100].valid := 1, [16].log_data[101].valid := 1, [16].log_data[102].valid := 1, [16].log_data[103].valid := 1, [16].log_data[104].valid := 1, [16].log_data[105].valid := 1, [16].log_data[106].valid := 1,
        [16].log_data[107].valid := 1, [16].log_data[108].valid := 1, [16].log_data[109].valid := 1, [16].log_data[110].valid := 1, [16].log_data[111].valid := 1, [16].log_data[112].valid := 1, [16].log_data[113].valid := 1, [16].log_data[114].valid := 1, [16].log_data[115].valid := 1, [16].log_data[116].valid := 1, [16].log_data[117].valid := 1, [16].log_data[118].valid := 1, [16].log_data[119].valid := 1, [16].log_data[120].valid := 1, [16].log_data[121].valid := 1, [16].log_data[122].valid := 1, [16].log_data[123].valid := 1, [16].log_data[124].valid := 1, [16].time.Year := 2023, [16].time.Month := 1, [16].time.Day := 13, [16].time.Hour := 19, [16].time.Minute := 59, [16].time.Second := 59, [17].log_data[0].min := 1.0, [17].log_data[0].max := 1.0, [17].log_data[0].total := 3600.0, [17].log_data[0].time := 3600.0, [17].log_data[0].valid := 1, [17].log_data[1].max := 1.0, [17].log_data[1].total := 552.751, [17].log_data[1].time := 3600.0, [17].log_data[1].minminute := 9, [17].log_data[1].valid := 1, [17].log_data[2].max := 1.0, [17].log_data[2].total := 551.5, [17].log_data[2].time := 3600.0, [17].log_data[2].valid := 1, [17].log_data[3].time := 3600.0, [17].log_data[3].valid := 1, [17].log_data[4].time := 3600.0, [17].log_data[4].valid := 1, [17].log_data[5].max := 1.0, [17].log_data[5].total := 249.0, [17].log_data[5].time := 3600.0, [17].log_data[5].maxminute := 2, [17].log_data[5].valid := 1, [17].log_data[6].time := 3600.0, [17].log_data[6].valid := 1, [17].log_data[7].time := 3600.0, [17].log_data[7].valid := 1, [17].log_data[8].max := 1.0, [17].log_data[8].total := 3363.249, [17].log_data[8].time := 3600.0, [17].log_data[8].maxminute := 3, [17].log_data[8].valid := 1, [17].log_data[9].max := 1.0, [17].log_data[9].total := 3359.749, [17].log_data[9].time := 3600.0, [17].log_data[9].maxminute := 4,
        [17].log_data[9].valid := 1, [17].log_data[10].min := 1.0, [17].log_data[10].max := 1.0, [17].log_data[10].total := 3600.0, [17].log_data[10].time := 3600.0, [17].log_data[10].valid := 1, [17].log_data[11].time := 3600.0, [17].log_data[11].valid := 1, [17].log_data[12].min := 1.0, [17].log_data[12].max := 1.0, [17].log_data[12].total := 3600.0, [17].log_data[12].time := 3600.0, [17].log_data[12].valid := 1, [17].log_data[13].min := 1.0, [17].log_data[13].max := 1.0, [17].log_data[13].total := 3600.0, [17].log_data[13].time := 3600.0, [17].log_data[13].valid := 1, [17].log_data[14].time := 3600.0, [17].log_data[14].valid := 1, [17].log_data[15].time := 3600.0, [17].log_data[15].valid := 1, [17].log_data[16].time := 3600.0, [17].log_data[16].valid := 1, [17].log_data[17].min := 1.0, [17].log_data[17].max := 1.0, [17].log_data[17].total := 3600.0, [17].log_data[17].time := 3600.0, [17].log_data[17].valid := 1, [17].log_data[18].time := 3600.0, [17].log_data[18].valid := 1, [17].log_data[19].time := 3600.0, [17].log_data[19].valid := 1, [17].log_data[20].time := 3600.0, [17].log_data[20].valid := 1, [17].log_data[21].min := 1.0, [17].log_data[21].max := 1.0, [17].log_data[21].total := 3600.0, [17].log_data[21].time := 3600.0, [17].log_data[21].valid := 1, [17].log_data[22].time := 3600.0, [17].log_data[22].valid := 1, [17].log_data[23].time := 3600.0, [17].log_data[23].valid := 1, [17].log_data[24].time := 3600.0, [17].log_data[24].valid := 1, [17].log_data[25].time := 3600.0, [17].log_data[25].valid := 1, [17].log_data[26].time := 3600.0, [17].log_data[26].valid := 1, [17].log_data[27].time := 3600.0, [17].log_data[27].valid := 1, [17].log_data[28].time := 3600.0, [17].log_data[28].valid := 1, [17].log_data[29].min := 1.0, [17].log_data[29].max := 1.0, [17].log_data[29].total := 3600.0, [17].log_data[29].time := 3600.0, [17].log_data[29].valid := 1, [17].log_data[30].min := 1.0,
        [17].log_data[30].max := 1.0, [17].log_data[30].total := 3600.0, [17].log_data[30].time := 3600.0, [17].log_data[30].valid := 1, [17].log_data[31].max := 1.0, [17].log_data[31].total := 1629.7471, [17].log_data[31].time := 3600.0, [17].log_data[31].maxminute := 5, [17].log_data[31].valid := 1, [17].log_data[32].max := 1.0, [17].log_data[32].total := 1197.498, [17].log_data[32].time := 3600.0, [17].log_data[32].maxminute := 4, [17].log_data[32].valid := 1, [17].log_data[33].time := 3600.0, [17].log_data[33].valid := 1, [17].log_data[34].time := 3600.0, [17].log_data[34].valid := 1, [17].log_data[35].max := 1.0, [17].log_data[35].total := 1391.998, [17].log_data[35].time := 3600.0, [17].log_data[35].maxminute := 4, [17].log_data[35].valid := 1, [17].log_data[36].max := 1.0, [17].log_data[36].total := 1519.2471, [17].log_data[36].time := 3600.0, [17].log_data[36].maxminute := 10, [17].log_data[36].valid := 1, [17].log_data[37].max := 7.5281005, [17].log_data[37].total := 3608.7566, [17].log_data[37].time := 3600.0, [17].log_data[37].minminute := 8, [17].log_data[37].valid := 1, [17].log_data[38].time := 3600.0, [17].log_data[38].valid := 1, [17].log_data[39].min := 0.9924686, [17].log_data[39].max := 1.0210879, [17].log_data[39].total := 3604.6392, [17].log_data[39].time := 3600.0, [17].log_data[39].minminute := 15, [17].log_data[39].maxminute := 6, [17].log_data[39].valid := 1, [17].log_data[40].min := 7.538759, [17].log_data[40].max := 7.603339, [17].log_data[40].total := 27278.28, [17].log_data[40].time := 3600.0, [17].log_data[40].minminute := 20, [17].log_data[40].maxminute := 29, [17].log_data[40].valid := 1, [17].log_data[41].min := 0.045309816, [17].log_data[41].max := 0.08123121, [17].log_data[41].total := 241.86339, [17].log_data[41].time := 3600.0, [17].log_data[41].minminute := 1, [17].log_data[41].maxminute := 12, [17].log_data[41].valid := 1, [17].log_data[42].min := 2.2922316, [17].log_data[42].max := 2.2985914, [17].log_data[42].total := 8263.747, [17].log_data[42].time := 3600.0,
        [17].log_data[42].minminute := 12, [17].log_data[42].maxminute := 53, [17].log_data[42].valid := 1, [17].log_data[43].min := -0.27999878, [17].log_data[43].max := -0.26000214, [17].log_data[43].total := -955.4761, [17].log_data[43].time := 3600.0, [17].log_data[43].valid := 1, [17].log_data[44].min := -0.30000305, [17].log_data[44].max := -0.27999878, [17].log_data[44].total := -1080.0812, [17].log_data[44].time := 3600.0, [17].log_data[44].maxminute := 16, [17].log_data[44].valid := 1, [17].log_data[45].time := 3600.0, [17].log_data[45].valid := 1, [17].log_data[46].time := 3600.0, [17].log_data[46].valid := 1, [17].log_data[47].time := 3600.0, [17].log_data[47].valid := 1, [17].log_data[48].min := 6.5810537, [17].log_data[48].max := 6.9765024, [17].log_data[48].total := 24235.36, [17].log_data[48].time := 3600.0, [17].log_data[48].minminute := 32, [17].log_data[48].maxminute := 8, [17].log_data[48].valid := 1, [17].log_data[49].min := 6.825411, [17].log_data[49].max := 9.474756, [17].log_data[49].total := 28874.186, [17].log_data[49].time := 3600.0, [17].log_data[49].minminute := 26, [17].log_data[49].maxminute := 2, [17].log_data[49].valid := 1, [17].log_data[50].min := 2.0504398, [17].log_data[50].max := 2.151137, [17].log_data[50].total := 7515.725, [17].log_data[50].time := 3600.0, [17].log_data[50].minminute := 57, [17].log_data[50].maxminute := 3, [17].log_data[50].valid := 1, [17].log_data[51].time := 3600.0, [17].log_data[51].valid := 1, [17].log_data[52].min := -4.1800003, [17].log_data[52].max := 0.11999512, [17].log_data[52].total := -7350.3125, [17].log_data[52].time := 3600.0, [17].log_data[52].minminute := 4, [17].log_data[52].maxminute := 5, [17].log_data[52].valid := 1, [17].log_data[53].min := -4.0, [17].log_data[53].max := 0.19999695, [17].log_data[53].total := -7005.8037, [17].log_data[53].time := 3600.0, [17].log_data[53].minminute := 4, [17].log_data[53].maxminute := 20, [17].log_data[53].valid := 1, [17].log_data[54].max := 0.5375, [17].log_data[54].total := 1117.7933, [17].log_data[54].time := 3600.0,
        [17].log_data[54].maxminute := 6, [17].log_data[54].valid := 1, [17].log_data[55].max := 0.533, [17].log_data[55].total := 1153.4188, [17].log_data[55].time := 3600.0, [17].log_data[55].maxminute := 4, [17].log_data[55].valid := 1, [17].log_data[56].min := 0.16024561, [17].log_data[56].max := 0.16067745, [17].log_data[56].total := 577.50134, [17].log_data[56].time := 3600.0, [17].log_data[56].minminute := 21, [17].log_data[56].maxminute := 55, [17].log_data[56].valid := 1, [17].log_data[57].min := 0.306679, [17].log_data[57].max := 0.30864188, [17].log_data[57].total := 1107.9426, [17].log_data[57].time := 3600.0, [17].log_data[57].minminute := 46, [17].log_data[57].maxminute := 10, [17].log_data[57].valid := 1, [17].log_data[58].time := 3600.0, [17].log_data[58].valid := 1, [17].log_data[59].time := 3600.0, [17].log_data[59].valid := 1, [17].log_data[60].valid := 1, [17].log_data[61].valid := 1, [17].log_data[62].valid := 1, [17].log_data[63].valid := 1, [17].log_data[64].valid := 1, [17].log_data[65].valid := 1, [17].log_data[66].valid := 1, [17].log_data[67].valid := 1, [17].log_data[68].valid := 1, [17].log_data[69].valid := 1, [17].log_data[70].valid := 1, [17].log_data[71].valid := 1, [17].log_data[72].valid := 1, [17].log_data[73].valid := 1, [17].log_data[74].valid := 1, [17].log_data[75].valid := 1, [17].log_data[76].valid := 1, [17].log_data[77].valid := 1, [17].log_data[78].valid := 1, [17].log_data[79].valid := 1, [17].log_data[80].valid := 1, [17].log_data[81].valid := 1, [17].log_data[82].valid := 1, [17].log_data[83].valid := 1, [17].log_data[84].valid := 1, [17].log_data[85].valid := 1, [17].log_data[86].valid := 1, [17].log_data[87].valid := 1, [17].log_data[88].valid := 1, [17].log_data[89].valid := 1, [17].log_data[90].valid := 1, [17].log_data[91].valid := 1, [17].log_data[92].valid := 1, [17].log_data[93].valid := 1, [17].log_data[94].valid := 1,
        [17].log_data[95].valid := 1, [17].log_data[96].valid := 1, [17].log_data[97].valid := 1, [17].log_data[98].valid := 1, [17].log_data[99].valid := 1, [17].log_data[100].valid := 1, [17].log_data[101].valid := 1, [17].log_data[102].valid := 1, [17].log_data[103].valid := 1, [17].log_data[104].valid := 1, [17].log_data[105].valid := 1, [17].log_data[106].valid := 1, [17].log_data[107].valid := 1, [17].log_data[108].valid := 1, [17].log_data[109].valid := 1, [17].log_data[110].valid := 1, [17].log_data[111].valid := 1, [17].log_data[112].valid := 1, [17].log_data[113].valid := 1, [17].log_data[114].valid := 1, [17].log_data[115].valid := 1, [17].log_data[116].valid := 1, [17].log_data[117].valid := 1, [17].log_data[118].valid := 1, [17].log_data[119].valid := 1, [17].log_data[120].valid := 1, [17].log_data[121].valid := 1, [17].log_data[122].valid := 1, [17].log_data[123].valid := 1, [17].log_data[124].valid := 1, [17].time.Year := 2023, [17].time.Month := 1, [17].time.Day := 13, [17].time.Hour := 20, [17].time.Minute := 59, [17].time.Second := 59, [18].log_data[0].min := 1.0, [18].log_data[0].max := 1.0, [18].log_data[0].total := 3600.0, [18].log_data[0].time := 3600.0, [18].log_data[0].valid := 1, [18].log_data[1].max := 1.0, [18].log_data[1].total := 569.5, [18].log_data[1].time := 3600.0, [18].log_data[1].maxminute := 15, [18].log_data[1].valid := 1, [18].log_data[2].max := 1.0, [18].log_data[2].total := 566.0, [18].log_data[2].time := 3600.0, [18].log_data[2].maxminute := 15, [18].log_data[2].valid := 1, [18].log_data[3].time := 3600.0, [18].log_data[3].valid := 1, [18].log_data[4].time := 3600.0, [18].log_data[4].valid := 1, [18].log_data[5].max := 1.0, [18].log_data[5].total := 233.5, [18].log_data[5].time := 3600.0, [18].log_data[5].maxminute := 18, [18].log_data[5].valid := 1,
        [18].log_data[6].time := 3600.0, [18].log_data[6].valid := 1, [18].log_data[7].time := 3600.0, [18].log_data[7].valid := 1, [18].log_data[8].min := 1.0, [18].log_data[8].max := 1.0, [18].log_data[8].total := 3600.0, [18].log_data[8].time := 3600.0, [18].log_data[8].valid := 1, [18].log_data[9].min := 1.0, [18].log_data[9].max := 1.0, [18].log_data[9].total := 3600.0, [18].log_data[9].time := 3600.0, [18].log_data[9].valid := 1, [18].log_data[10].min := 1.0, [18].log_data[10].max := 1.0, [18].log_data[10].total := 3600.0, [18].log_data[10].time := 3600.0, [18].log_data[10].valid := 1, [18].log_data[11].time := 3600.0, [18].log_data[11].valid := 1, [18].log_data[12].min := 1.0, [18].log_data[12].max := 1.0, [18].log_data[12].total := 3600.0, [18].log_data[12].time := 3600.0, [18].log_data[12].valid := 1, [18].log_data[13].min := 1.0, [18].log_data[13].max := 1.0, [18].log_data[13].total := 3600.0, [18].log_data[13].time := 3600.0, [18].log_data[13].valid := 1, [18].log_data[14].time := 3600.0, [18].log_data[14].valid := 1, [18].log_data[15].time := 3600.0, [18].log_data[15].valid := 1, [18].log_data[16].time := 3600.0, [18].log_data[16].valid := 1, [18].log_data[17].min := 1.0, [18].log_data[17].max := 1.0, [18].log_data[17].total := 3600.0, [18].log_data[17].time := 3600.0, [18].log_data[17].valid := 1, [18].log_data[18].time := 3600.0, [18].log_data[18].valid := 1, [18].log_data[19].time := 3600.0, [18].log_data[19].valid := 1, [18].log_data[20].time := 3600.0, [18].log_data[20].valid := 1, [18].log_data[21].min := 1.0, [18].log_data[21].max := 1.0, [18].log_data[21].total := 3600.0, [18].log_data[21].time := 3600.0, [18].log_data[21].valid := 1, [18].log_data[22].time := 3600.0, [18].log_data[22].valid := 1, [18].log_data[23].time := 3600.0, [18].log_data[23].valid := 1, [18].log_data[24].time := 3600.0, [18].log_data[24].valid := 1, [18].log_data[25].time := 3600.0,
        [18].log_data[25].valid := 1, [18].log_data[26].time := 3600.0, [18].log_data[26].valid := 1, [18].log_data[27].time := 3600.0, [18].log_data[27].valid := 1, [18].log_data[28].time := 3600.0, [18].log_data[28].valid := 1, [18].log_data[29].min := 1.0, [18].log_data[29].max := 1.0, [18].log_data[29].total := 3600.0, [18].log_data[29].time := 3600.0, [18].log_data[29].valid := 1, [18].log_data[30].min := 1.0, [18].log_data[30].max := 1.0, [18].log_data[30].total := 3600.0, [18].log_data[30].time := 3600.0, [18].log_data[30].valid := 1, [18].log_data[31].max := 1.0, [18].log_data[31].total := 1617.498, [18].log_data[31].time := 3600.0, [18].log_data[31].maxminute := 9, [18].log_data[31].valid := 1, [18].log_data[32].max := 1.0, [18].log_data[32].total := 1541.749, [18].log_data[32].time := 3600.0, [18].log_data[32].minminute := 7, [18].log_data[32].valid := 1, [18].log_data[33].time := 3600.0, [18].log_data[33].valid := 1, [18].log_data[34].time := 3600.0, [18].log_data[34].valid := 1, [18].log_data[35].max := 1.0, [18].log_data[35].total := 1629.7471, [18].log_data[35].time := 3600.0, [18].log_data[35].maxminute := 3, [18].log_data[35].valid := 1, [18].log_data[36].max := 1.0, [18].log_data[36].total := 1440.749, [18].log_data[36].time := 3600.0, [18].log_data[36].minminute := 1, [18].log_data[36].valid := 1, [18].log_data[37].max := 7.213641, [18].log_data[37].total := 3574.8318, [18].log_data[37].time := 3600.0, [18].log_data[37].maxminute := 16, [18].log_data[37].valid := 1, [18].log_data[38].time := 3600.0, [18].log_data[38].valid := 1, [18].log_data[39].min := 0.9939996, [18].log_data[39].max := 1.0213233, [18].log_data[39].total := 3608.2468, [18].log_data[39].time := 3600.0, [18].log_data[39].minminute := 8, [18].log_data[39].maxminute := 18, [18].log_data[39].valid := 1, [18].log_data[40].min := 7.560194, [18].log_data[40].max := 7.5849276, [18].log_data[40].total := 27280.312, [18].log_data[40].time := 3600.0, [18].log_data[40].minminute := 16,
        [18].log_data[40].maxminute := 40, [18].log_data[40].valid := 1, [18].log_data[41].min := 0.03804712, [18].log_data[41].max := 0.076127686, [18].log_data[41].total := 187.5313, [18].log_data[41].time := 3600.0, [18].log_data[41].minminute := 59, [18].log_data[41].valid := 1, [18].log_data[42].min := 2.2927027, [18].log_data[42].max := 2.2978847, [18].log_data[42].total := 8263.7295, [18].log_data[42].time := 3600.0, [18].log_data[42].minminute := 50, [18].log_data[42].maxminute := 16, [18].log_data[42].valid := 1, [18].log_data[43].min := -0.27999878, [18].log_data[43].max := -0.26000214, [18].log_data[43].total := -940.68066, [18].log_data[43].time := 3600.0, [18].log_data[43].valid := 1, [18].log_data[44].min := -0.30000305, [18].log_data[44].max := -0.27999878, [18].log_data[44].total := -1079.9103, [18].log_data[44].time := 3600.0, [18].log_data[44].maxminute := 18, [18].log_data[44].valid := 1, [18].log_data[45].time := 3600.0, [18].log_data[45].valid := 1, [18].log_data[46].time := 3600.0, [18].log_data[46].valid := 1, [18].log_data[47].time := 3600.0, [18].log_data[47].valid := 1, [18].log_data[48].min := 6.5810537, [18].log_data[48].max := 6.969357, [18].log_data[48].total := 24217.393, [18].log_data[48].time := 3600.0, [18].log_data[48].minminute := 48, [18].log_data[48].maxminute := 24, [18].log_data[48].valid := 1, [18].log_data[49].min := 6.9027495, [18].log_data[49].max := 9.474756, [18].log_data[49].total := 29578.166, [18].log_data[49].time := 3600.0, [18].log_data[49].minminute := 43, [18].log_data[49].maxminute := 18, [18].log_data[49].valid := 1, [18].log_data[50].min := 2.022056, [18].log_data[50].max := 2.1280534, [18].log_data[50].total := 7496.864, [18].log_data[50].time := 3600.0, [18].log_data[50].minminute := 18, [18].log_data[50].maxminute := 27, [18].log_data[50].valid := 1, [18].log_data[51].time := 3600.0, [18].log_data[51].valid := 1, [18].log_data[52].min := -2.840004, [18].log_data[52].max := 0.11999512, [18].log_data[52].total := -7798.5522, [18].log_data[52].time := 3600.0, [18].log_data[52].minminute := 30,
        [18].log_data[52].maxminute := 7, [18].log_data[52].valid := 1, [18].log_data[53].min := -2.4800034, [18].log_data[53].max := 0.22000122, [18].log_data[53].total := -6968.358, [18].log_data[53].time := 3600.0, [18].log_data[53].minminute := 41, [18].log_data[53].maxminute := 34, [18].log_data[53].valid := 1, [18].log_data[54].max := 0.53, [18].log_data[54].total := 1254.4773, [18].log_data[54].time := 3600.0, [18].log_data[54].minminute := 7, [18].log_data[54].maxminute := 9, [18].log_data[54].valid := 1, [18].log_data[55].max := 0.523, [18].log_data[55].total := 1217.2968, [18].log_data[55].time := 3600.0, [18].log_data[55].minminute := 1, [18].log_data[55].maxminute := 34, [18].log_data[55].valid := 1, [18].log_data[56].min := 0.16024561, [18].log_data[56].max := 0.16063818, [18].log_data[56].total := 577.48016, [18].log_data[56].time := 3600.0, [18].log_data[56].minminute := 49, [18].log_data[56].maxminute := 1, [18].log_data[56].valid := 1, [18].log_data[57].min := 0.3051479, [18].log_data[57].max := 0.3070716, [18].log_data[57].total := 1103.7035, [18].log_data[57].time := 3600.0, [18].log_data[57].minminute := 55, [18].log_data[57].maxminute := 3, [18].log_data[57].valid := 1, [18].log_data[58].time := 3600.0, [18].log_data[58].valid := 1, [18].log_data[59].time := 3600.0, [18].log_data[59].valid := 1, [18].log_data[60].valid := 1, [18].log_data[61].valid := 1, [18].log_data[62].valid := 1, [18].log_data[63].valid := 1, [18].log_data[64].valid := 1, [18].log_data[65].valid := 1, [18].log_data[66].valid := 1, [18].log_data[67].valid := 1, [18].log_data[68].valid := 1, [18].log_data[69].valid := 1, [18].log_data[70].valid := 1, [18].log_data[71].valid := 1, [18].log_data[72].valid := 1, [18].log_data[73].valid := 1, [18].log_data[74].valid := 1, [18].log_data[75].valid := 1, [18].log_data[76].valid := 1, [18].log_data[77].valid := 1, [18].log_data[78].valid := 1, [18].log_data[79].valid := 1, [18].log_data[80].valid := 1,
        [18].log_data[81].valid := 1, [18].log_data[82].valid := 1, [18].log_data[83].valid := 1, [18].log_data[84].valid := 1, [18].log_data[85].valid := 1, [18].log_data[86].valid := 1, [18].log_data[87].valid := 1, [18].log_data[88].valid := 1, [18].log_data[89].valid := 1, [18].log_data[90].valid := 1, [18].log_data[91].valid := 1, [18].log_data[92].valid := 1, [18].log_data[93].valid := 1, [18].log_data[94].valid := 1, [18].log_data[95].valid := 1, [18].log_data[96].valid := 1, [18].log_data[97].valid := 1, [18].log_data[98].valid := 1, [18].log_data[99].valid := 1, [18].log_data[100].valid := 1, [18].log_data[101].valid := 1, [18].log_data[102].valid := 1, [18].log_data[103].valid := 1, [18].log_data[104].valid := 1, [18].log_data[105].valid := 1, [18].log_data[106].valid := 1, [18].log_data[107].valid := 1, [18].log_data[108].valid := 1, [18].log_data[109].valid := 1, [18].log_data[110].valid := 1, [18].log_data[111].valid := 1, [18].log_data[112].valid := 1, [18].log_data[113].valid := 1, [18].log_data[114].valid := 1, [18].log_data[115].valid := 1, [18].log_data[116].valid := 1, [18].log_data[117].valid := 1, [18].log_data[118].valid := 1, [18].log_data[119].valid := 1, [18].log_data[120].valid := 1, [18].log_data[121].valid := 1, [18].log_data[122].valid := 1, [18].log_data[123].valid := 1, [18].log_data[124].valid := 1, [18].time.Year := 2023, [18].time.Month := 1, [18].time.Day := 13, [18].time.Hour := 21, [18].time.Minute := 59, [18].time.Second := 59, [19].log_data[0].min := 1.0, [19].log_data[0].max := 1.0, [19].log_data[0].total := 3600.0, [19].log_data[0].time := 3600.0, [19].log_data[0].valid := 1, [19].log_data[1].max := 1.0, [19].log_data[1].total := 552.0, [19].log_data[1].time := 3600.0, [19].log_data[1].maxminute := 32, [19].log_data[1].valid := 1,
        [19].log_data[2].max := 1.0, [19].log_data[2].total := 548.5, [19].log_data[2].time := 3600.0, [19].log_data[2].maxminute := 32, [19].log_data[2].valid := 1, [19].log_data[3].time := 3600.0, [19].log_data[3].valid := 1, [19].log_data[4].time := 3600.0, [19].log_data[4].valid := 1, [19].log_data[5].max := 1.0, [19].log_data[5].total := 239.0, [19].log_data[5].time := 3600.0, [19].log_data[5].maxminute := 34, [19].log_data[5].valid := 1, [19].log_data[6].time := 3600.0, [19].log_data[6].valid := 1, [19].log_data[7].time := 3600.0, [19].log_data[7].valid := 1, [19].log_data[8].min := 1.0, [19].log_data[8].max := 1.0, [19].log_data[8].total := 3600.0, [19].log_data[8].time := 3600.0, [19].log_data[8].valid := 1, [19].log_data[9].min := 1.0, [19].log_data[9].max := 1.0, [19].log_data[9].total := 3600.0, [19].log_data[9].time := 3600.0, [19].log_data[9].valid := 1, [19].log_data[10].min := 1.0, [19].log_data[10].max := 1.0, [19].log_data[10].total := 3600.0, [19].log_data[10].time := 3600.0, [19].log_data[10].valid := 1, [19].log_data[11].time := 3600.0, [19].log_data[11].valid := 1, [19].log_data[12].min := 1.0, [19].log_data[12].max := 1.0, [19].log_data[12].total := 3600.0, [19].log_data[12].time := 3600.0, [19].log_data[12].valid := 1, [19].log_data[13].min := 1.0, [19].log_data[13].max := 1.0, [19].log_data[13].total := 3600.0, [19].log_data[13].time := 3600.0, [19].log_data[13].valid := 1, [19].log_data[14].time := 3600.0, [19].log_data[14].valid := 1, [19].log_data[15].time := 3600.0, [19].log_data[15].valid := 1, [19].log_data[16].time := 3600.0, [19].log_data[16].valid := 1, [19].log_data[17].min := 1.0, [19].log_data[17].max := 1.0, [19].log_data[17].total := 3600.0, [19].log_data[17].time := 3600.0, [19].log_data[17].valid := 1, [19].log_data[18].time := 3600.0, [19].log_data[18].valid := 1, [19].log_data[19].time := 3600.0, [19].log_data[19].valid := 1,
        [19].log_data[20].time := 3600.0, [19].log_data[20].valid := 1, [19].log_data[21].min := 1.0, [19].log_data[21].max := 1.0, [19].log_data[21].total := 3600.0, [19].log_data[21].time := 3600.0, [19].log_data[21].valid := 1, [19].log_data[22].time := 3600.0, [19].log_data[22].valid := 1, [19].log_data[23].time := 3600.0, [19].log_data[23].valid := 1, [19].log_data[24].time := 3600.0, [19].log_data[24].valid := 1, [19].log_data[25].time := 3600.0, [19].log_data[25].valid := 1, [19].log_data[26].time := 3600.0, [19].log_data[26].valid := 1, [19].log_data[27].time := 3600.0, [19].log_data[27].valid := 1, [19].log_data[28].time := 3600.0, [19].log_data[28].valid := 1, [19].log_data[29].min := 1.0, [19].log_data[29].max := 1.0, [19].log_data[29].total := 3600.0, [19].log_data[29].time := 3600.0, [19].log_data[29].valid := 1, [19].log_data[30].min := 1.0, [19].log_data[30].max := 1.0, [19].log_data[30].total := 3600.0, [19].log_data[30].time := 3600.0, [19].log_data[30].valid := 1, [19].log_data[31].max := 1.0, [19].log_data[31].total := 1440.498, [19].log_data[31].time := 3600.0, [19].log_data[31].valid := 1, [19].log_data[32].max := 1.0, [19].log_data[32].total := 1629.998, [19].log_data[32].time := 3600.0, [19].log_data[32].maxminute := 1, [19].log_data[32].valid := 1, [19].log_data[33].time := 3600.0, [19].log_data[33].valid := 1, [19].log_data[34].time := 3600.0, [19].log_data[34].valid := 1, [19].log_data[35].max := 1.0, [19].log_data[35].total := 1629.7471, [19].log_data[35].time := 3600.0, [19].log_data[35].maxminute := 6, [19].log_data[35].valid := 1, [19].log_data[36].max := 1.0, [19].log_data[36].total := 1440.7471, [19].log_data[36].time := 3600.0, [19].log_data[36].minminute := 4, [19].log_data[36].valid := 1, [19].log_data[37].max := 7.5065084, [19].log_data[37].total := 3608.1692, [19].log_data[37].time := 3600.0, [19].log_data[37].maxminute := 33, [19].log_data[37].valid := 1, [19].log_data[38].time := 3600.0,
        [19].log_data[38].valid := 1, [19].log_data[39].min := 0.99494183, [19].log_data[39].max := 1.0213233, [19].log_data[39].total := 3609.4363, [19].log_data[39].time := 3600.0, [19].log_data[39].minminute := 58, [19].log_data[39].maxminute := 38, [19].log_data[39].valid := 1, [19].log_data[40].min := 7.551675, [19].log_data[40].max := 7.586301, [19].log_data[40].total := 27282.455, [19].log_data[40].time := 3600.0, [19].log_data[40].minminute := 51, [19].log_data[40].maxminute := 57, [19].log_data[40].valid := 1, [19].log_data[41].min := 0.035102785, [19].log_data[41].max := 0.06906128, [19].log_data[41].total := 175.25644, [19].log_data[41].time := 3600.0, [19].log_data[41].minminute := 31, [19].log_data[41].maxminute := 41, [19].log_data[41].valid := 1, [19].log_data[42].min := 2.292585, [19].log_data[42].max := 2.2976491, [19].log_data[42].total := 8263.566, [19].log_data[42].time := 3600.0, [19].log_data[42].minminute := 5, [19].log_data[42].maxminute := 34, [19].log_data[42].valid := 1, [19].log_data[43].min := -0.27999878, [19].log_data[43].max := -0.26000214, [19].log_data[43].total := -938.3509, [19].log_data[43].time := 3600.0, [19].log_data[43].valid := 1, [19].log_data[44].min := -0.30000305, [19].log_data[44].max := -0.27999878, [19].log_data[44].total := -1079.976, [19].log_data[44].time := 3600.0, [19].log_data[44].maxminute := 6, [19].log_data[44].valid := 1, [19].log_data[45].time := 3600.0, [19].log_data[45].valid := 1, [19].log_data[46].time := 3600.0, [19].log_data[46].valid := 1, [19].log_data[47].time := 3600.0, [19].log_data[47].valid := 1, [19].log_data[48].min := 6.620901, [19].log_data[48].max := 6.959464, [19].log_data[48].total := 24378.285, [19].log_data[48].time := 3600.0, [19].log_data[48].minminute := 59, [19].log_data[48].maxminute := 41, [19].log_data[48].valid := 1, [19].log_data[49].min := 6.9127607, [19].log_data[49].max := 9.497918, [19].log_data[49].total := 30948.342, [19].log_data[49].time := 3600.0, [19].log_data[49].minminute := 58, [19].log_data[49].maxminute := 34, [19].log_data[49].valid := 1,
        [19].log_data[50].min := 2.0348935, [19].log_data[50].max := 2.1437175, [19].log_data[50].total := 7513.7207, [19].log_data[50].time := 3600.0, [19].log_data[50].minminute := 34, [19].log_data[50].maxminute := 41, [19].log_data[50].valid := 1, [19].log_data[51].time := 3600.0, [19].log_data[51].valid := 1, [19].log_data[52].min := -2.9199982, [19].log_data[52].max := 0.11999512, [19].log_data[52].total := -7523.0312, [19].log_data[52].time := 3600.0, [19].log_data[52].minminute := 12, [19].log_data[52].valid := 1, [19].log_data[53].min := -2.4800034, [19].log_data[53].max := 0.19999695, [19].log_data[53].total := -6942.6807, [19].log_data[53].time := 3600.0, [19].log_data[53].minminute := 48, [19].log_data[53].maxminute := 16, [19].log_data[53].valid := 1, [19].log_data[54].max := 0.5445, [19].log_data[54].total := 1217.1826, [19].log_data[54].time := 3600.0, [19].log_data[54].maxminute := 22, [19].log_data[54].valid := 1, [19].log_data[55].max := 0.542, [19].log_data[55].total := 1217.2527, [19].log_data[55].time := 3600.0, [19].log_data[55].minminute := 5, [19].log_data[55].maxminute := 48, [19].log_data[55].valid := 1, [19].log_data[56].min := 0.16028486, [19].log_data[56].max := 0.16067745, [19].log_data[56].total := 577.5408, [19].log_data[56].time := 3600.0, [19].log_data[56].minminute := 3, [19].log_data[56].maxminute := 20, [19].log_data[56].valid := 1, [19].log_data[57].min := 0.30503014, [19].log_data[57].max := 0.30550122, [19].log_data[57].total := 1098.78, [19].log_data[57].time := 3600.0, [19].log_data[57].minminute := 16, [19].log_data[57].maxminute := 21, [19].log_data[57].valid := 1, [19].log_data[58].time := 3600.0, [19].log_data[58].valid := 1, [19].log_data[59].time := 3600.0, [19].log_data[59].valid := 1, [19].log_data[60].valid := 1, [19].log_data[61].valid := 1, [19].log_data[62].valid := 1, [19].log_data[63].valid := 1, [19].log_data[64].valid := 1, [19].log_data[65].valid := 1, [19].log_data[66].valid := 1, [19].log_data[67].valid := 1, [19].log_data[68].valid := 1,
        [19].log_data[69].valid := 1, [19].log_data[70].valid := 1, [19].log_data[71].valid := 1, [19].log_data[72].valid := 1, [19].log_data[73].valid := 1, [19].log_data[74].valid := 1, [19].log_data[75].valid := 1, [19].log_data[76].valid := 1, [19].log_data[77].valid := 1, [19].log_data[78].valid := 1, [19].log_data[79].valid := 1, [19].log_data[80].valid := 1, [19].log_data[81].valid := 1, [19].log_data[82].valid := 1, [19].log_data[83].valid := 1, [19].log_data[84].valid := 1, [19].log_data[85].valid := 1, [19].log_data[86].valid := 1, [19].log_data[87].valid := 1, [19].log_data[88].valid := 1, [19].log_data[89].valid := 1, [19].log_data[90].valid := 1, [19].log_data[91].valid := 1, [19].log_data[92].valid := 1, [19].log_data[93].valid := 1, [19].log_data[94].valid := 1, [19].log_data[95].valid := 1, [19].log_data[96].valid := 1, [19].log_data[97].valid := 1, [19].log_data[98].valid := 1, [19].log_data[99].valid := 1, [19].log_data[100].valid := 1, [19].log_data[101].valid := 1, [19].log_data[102].valid := 1, [19].log_data[103].valid := 1, [19].log_data[104].valid := 1, [19].log_data[105].valid := 1, [19].log_data[106].valid := 1, [19].log_data[107].valid := 1, [19].log_data[108].valid := 1, [19].log_data[109].valid := 1, [19].log_data[110].valid := 1, [19].log_data[111].valid := 1, [19].log_data[112].valid := 1, [19].log_data[113].valid := 1, [19].log_data[114].valid := 1, [19].log_data[115].valid := 1, [19].log_data[116].valid := 1, [19].log_data[117].valid := 1, [19].log_data[118].valid := 1, [19].log_data[119].valid := 1, [19].log_data[120].valid := 1, [19].log_data[121].valid := 1, [19].log_data[122].valid := 1, [19].log_data[123].valid := 1, [19].log_data[124].valid := 1, [19].time.Year := 2023, [19].time.Month := 1, [19].time.Day := 13, [19].time.Hour := 22,
        [19].time.Minute := 59, [19].time.Second := 59, [20].log_data[0].min := 1.0, [20].log_data[0].max := 1.0, [20].log_data[0].total := 3600.0, [20].log_data[0].time := 3600.0, [20].log_data[0].valid := 1, [20].log_data[1].time := 3600.0, [20].log_data[1].valid := 1, [20].log_data[2].time := 3600.0, [20].log_data[2].valid := 1, [20].log_data[3].time := 3600.0, [20].log_data[3].valid := 1, [20].log_data[4].time := 3600.0, [20].log_data[4].valid := 1, [20].log_data[5].time := 3600.0, [20].log_data[5].valid := 1, [20].log_data[6].time := 3600.0, [20].log_data[6].valid := 1, [20].log_data[7].time := 3600.0, [20].log_data[7].valid := 1, [20].log_data[8].min := 1.0, [20].log_data[8].max := 1.0, [20].log_data[8].total := 3600.0, [20].log_data[8].time := 3600.0, [20].log_data[8].valid := 1, [20].log_data[9].min := 1.0, [20].log_data[9].max := 1.0, [20].log_data[9].total := 3600.0, [20].log_data[9].time := 3600.0, [20].log_data[9].valid := 1, [20].log_data[10].min := 1.0, [20].log_data[10].max := 1.0, [20].log_data[10].total := 3600.0, [20].log_data[10].time := 3600.0, [20].log_data[10].valid := 1, [20].log_data[11].time := 3600.0, [20].log_data[11].valid := 1, [20].log_data[12].min := 1.0, [20].log_data[12].max := 1.0, [20].log_data[12].total := 3600.0, [20].log_data[12].time := 3600.0, [20].log_data[12].valid := 1, [20].log_data[13].min := 1.0, [20].log_data[13].max := 1.0, [20].log_data[13].total := 3600.0, [20].log_data[13].time := 3600.0, [20].log_data[13].valid := 1, [20].log_data[14].time := 3600.0, [20].log_data[14].valid := 1, [20].log_data[15].time := 3600.0, [20].log_data[15].valid := 1, [20].log_data[16].time := 3600.0, [20].log_data[16].valid := 1, [20].log_data[17].min := 1.0, [20].log_data[17].max := 1.0, [20].log_data[17].total := 3600.0, [20].log_data[17].time := 3600.0, [20].log_data[17].valid := 1, [20].log_data[18].time := 3600.0,
        [20].log_data[18].valid := 1, [20].log_data[19].time := 3600.0, [20].log_data[19].valid := 1, [20].log_data[20].time := 3600.0, [20].log_data[20].valid := 1, [20].log_data[21].min := 1.0, [20].log_data[21].max := 1.0, [20].log_data[21].total := 3600.0, [20].log_data[21].time := 3600.0, [20].log_data[21].valid := 1, [20].log_data[22].time := 3600.0, [20].log_data[22].valid := 1, [20].log_data[23].time := 3600.0, [20].log_data[23].valid := 1, [20].log_data[24].time := 3600.0, [20].log_data[24].valid := 1, [20].log_data[25].time := 3600.0, [20].log_data[25].valid := 1, [20].log_data[26].time := 3600.0, [20].log_data[26].valid := 1, [20].log_data[27].time := 3600.0, [20].log_data[27].valid := 1, [20].log_data[28].time := 3600.0, [20].log_data[28].valid := 1, [20].log_data[29].min := 1.0, [20].log_data[29].max := 1.0, [20].log_data[29].total := 3600.0, [20].log_data[29].time := 3600.0, [20].log_data[29].valid := 1, [20].log_data[30].min := 1.0, [20].log_data[30].max := 1.0, [20].log_data[30].total := 3600.0, [20].log_data[30].time := 3600.0, [20].log_data[30].valid := 1, [20].log_data[31].max := 1.0, [20].log_data[31].total := 1440.7471, [20].log_data[31].time := 3600.0, [20].log_data[31].minminute := 3, [20].log_data[31].valid := 1, [20].log_data[32].max := 1.0, [20].log_data[32].total := 1629.998, [20].log_data[32].time := 3600.0, [20].log_data[32].maxminute := 4, [20].log_data[32].valid := 1, [20].log_data[33].time := 3600.0, [20].log_data[33].valid := 1, [20].log_data[34].time := 3600.0, [20].log_data[34].valid := 1, [20].log_data[35].max := 1.0, [20].log_data[35].total := 1583.7471, [20].log_data[35].time := 3600.0, [20].log_data[35].maxminute := 9, [20].log_data[35].valid := 1, [20].log_data[36].max := 1.0, [20].log_data[36].total := 1574.998, [20].log_data[36].time := 3600.0, [20].log_data[36].minminute := 8, [20].log_data[36].valid := 1, [20].log_data[37].time := 3600.0, [20].log_data[37].valid := 1,
        [20].log_data[38].time := 3600.0, [20].log_data[38].valid := 1, [20].log_data[39].min := 0.9951773, [20].log_data[39].max := 1.006366, [20].log_data[39].total := 3604.6382, [20].log_data[39].time := 3600.0, [20].log_data[39].minminute := 43, [20].log_data[39].maxminute := 36, [20].log_data[39].valid := 1, [20].log_data[40].min := 7.548927, [20].log_data[40].max := 7.592072, [20].log_data[40].total := 27272.928, [20].log_data[40].time := 3600.0, [20].log_data[40].minminute := 46, [20].log_data[40].maxminute := 24, [20].log_data[40].valid := 1, [20].log_data[41].min := 0.03412134, [20].log_data[41].max := 0.056694824, [20].log_data[41].total := 162.04822, [20].log_data[41].time := 3600.0, [20].log_data[41].minminute := 33, [20].log_data[41].maxminute := 7, [20].log_data[41].valid := 1, [20].log_data[42].min := 2.2917604, [20].log_data[42].max := 2.2978847, [20].log_data[42].total := 8263.566, [20].log_data[42].time := 3600.0, [20].log_data[42].minminute := 21, [20].log_data[42].maxminute := 3, [20].log_data[42].valid := 1, [20].log_data[43].min := -0.27999878, [20].log_data[43].max := -0.26000214, [20].log_data[43].total := -936.994, [20].log_data[43].time := 3600.0, [20].log_data[43].minminute := 1, [20].log_data[43].valid := 1, [20].log_data[44].min := -0.30000305, [20].log_data[44].max := -0.27999878, [20].log_data[44].total := -1077.8058, [20].log_data[44].time := 3600.0, [20].log_data[44].maxminute := 1, [20].log_data[44].valid := 1, [20].log_data[45].time := 3600.0, [20].log_data[45].valid := 1, [20].log_data[46].time := 3600.0, [20].log_data[46].valid := 1, [20].log_data[47].time := 3600.0, [20].log_data[47].valid := 1, [20].log_data[48].min := 6.58655, [20].log_data[48].max := 6.78716, [20].log_data[48].total := 24238.863, [20].log_data[48].time := 3600.0, [20].log_data[48].minminute := 5, [20].log_data[48].maxminute := 20, [20].log_data[48].valid := 1, [20].log_data[49].min := 6.894702, [20].log_data[49].max := 9.532858, [20].log_data[49].total := 31485.088, [20].log_data[49].time := 3600.0, [20].log_data[49].maxminute := 59,
        [20].log_data[49].valid := 1, [20].log_data[50].min := 2.0378377, [20].log_data[50].max := 2.125109, [20].log_data[50].total := 7495.5923, [20].log_data[50].time := 3600.0, [20].log_data[50].minminute := 59, [20].log_data[50].valid := 1, [20].log_data[51].time := 3600.0, [20].log_data[51].valid := 1, [20].log_data[52].min := -2.840004, [20].log_data[52].max := 0.13999939, [20].log_data[52].total := -7512.854, [20].log_data[52].time := 3600.0, [20].log_data[52].minminute := 4, [20].log_data[52].maxminute := 56, [20].log_data[52].valid := 1, [20].log_data[53].min := -2.4600067, [20].log_data[53].max := 0.22000122, [20].log_data[53].total := -7190.9097, [20].log_data[53].time := 3600.0, [20].log_data[53].minminute := 53, [20].log_data[53].maxminute := 9, [20].log_data[53].valid := 1, [20].log_data[54].max := 0.538, [20].log_data[54].total := 1217.4739, [20].log_data[54].time := 3600.0, [20].log_data[54].minminute := 3, [20].log_data[54].maxminute := 4, [20].log_data[54].valid := 1, [20].log_data[55].max := 0.5165, [20].log_data[55].total := 1254.2198, [20].log_data[55].time := 3600.0, [20].log_data[55].minminute := 8, [20].log_data[55].maxminute := 51, [20].log_data[55].valid := 1, [20].log_data[56].min := 0.16020635, [20].log_data[56].max := 0.16063818, [20].log_data[56].total := 577.4556, [20].log_data[56].time := 3600.0, [20].log_data[56].minminute := 10, [20].log_data[56].maxminute := 1, [20].log_data[56].valid := 1, [20].log_data[57].min := 0.30381313, [20].log_data[57].max := 0.3054227, [20].log_data[57].total := 1094.8633, [20].log_data[57].time := 3600.0, [20].log_data[57].minminute := 19, [20].log_data[57].valid := 1, [20].log_data[58].time := 3600.0, [20].log_data[58].valid := 1, [20].log_data[59].time := 3600.0, [20].log_data[59].valid := 1, [20].log_data[60].valid := 1, [20].log_data[61].valid := 1, [20].log_data[62].valid := 1, [20].log_data[63].valid := 1, [20].log_data[64].valid := 1, [20].log_data[65].valid := 1, [20].log_data[66].valid := 1, [20].log_data[67].valid := 1,
        [20].log_data[68].valid := 1, [20].log_data[69].valid := 1, [20].log_data[70].valid := 1, [20].log_data[71].valid := 1, [20].log_data[72].valid := 1, [20].log_data[73].valid := 1, [20].log_data[74].valid := 1, [20].log_data[75].valid := 1, [20].log_data[76].valid := 1, [20].log_data[77].valid := 1, [20].log_data[78].valid := 1, [20].log_data[79].valid := 1, [20].log_data[80].valid := 1, [20].log_data[81].valid := 1, [20].log_data[82].valid := 1, [20].log_data[83].valid := 1, [20].log_data[84].valid := 1, [20].log_data[85].valid := 1, [20].log_data[86].valid := 1, [20].log_data[87].valid := 1, [20].log_data[88].valid := 1, [20].log_data[89].valid := 1, [20].log_data[90].valid := 1, [20].log_data[91].valid := 1, [20].log_data[92].valid := 1, [20].log_data[93].valid := 1, [20].log_data[94].valid := 1, [20].log_data[95].valid := 1, [20].log_data[96].valid := 1, [20].log_data[97].valid := 1, [20].log_data[98].valid := 1, [20].log_data[99].valid := 1, [20].log_data[100].valid := 1, [20].log_data[101].valid := 1, [20].log_data[102].valid := 1, [20].log_data[103].valid := 1, [20].log_data[104].valid := 1, [20].log_data[105].valid := 1, [20].log_data[106].valid := 1, [20].log_data[107].valid := 1, [20].log_data[108].valid := 1, [20].log_data[109].valid := 1, [20].log_data[110].valid := 1, [20].log_data[111].valid := 1, [20].log_data[112].valid := 1, [20].log_data[113].valid := 1, [20].log_data[114].valid := 1, [20].log_data[115].valid := 1, [20].log_data[116].valid := 1, [20].log_data[117].valid := 1, [20].log_data[118].valid := 1, [20].log_data[119].valid := 1, [20].log_data[120].valid := 1, [20].log_data[121].valid := 1, [20].log_data[122].valid := 1, [20].log_data[123].valid := 1, [20].log_data[124].valid := 1, [20].time.Year := 2023, [20].time.Month := 1, [20].time.Day := 13,
        [20].time.Hour := 23, [20].time.Minute := 59, [20].time.Second := 59, [21].log_data[0].min := 1.0, [21].log_data[0].max := 1.0, [21].log_data[0].total := 3599.5, [21].log_data[0].time := 3599.5, [21].log_data[0].valid := 1, [21].log_data[1].max := 1.0, [21].log_data[1].total := 558.0, [21].log_data[1].time := 3599.5, [21].log_data[1].maxminute := 8, [21].log_data[1].valid := 1, [21].log_data[2].max := 1.0, [21].log_data[2].total := 554.5, [21].log_data[2].time := 3599.5, [21].log_data[2].maxminute := 8, [21].log_data[2].valid := 1, [21].log_data[3].time := 3599.5, [21].log_data[3].valid := 1, [21].log_data[4].time := 3599.5, [21].log_data[4].valid := 1, [21].log_data[5].max := 1.0, [21].log_data[5].total := 235.5, [21].log_data[5].time := 3599.5, [21].log_data[5].maxminute := 10, [21].log_data[5].valid := 1, [21].log_data[6].time := 3599.5, [21].log_data[6].valid := 1, [21].log_data[7].time := 3599.5, [21].log_data[7].valid := 1, [21].log_data[8].min := 1.0, [21].log_data[8].max := 1.0, [21].log_data[8].total := 3599.5, [21].log_data[8].time := 3599.5, [21].log_data[8].valid := 1, [21].log_data[9].min := 1.0, [21].log_data[9].max := 1.0, [21].log_data[9].total := 3599.5, [21].log_data[9].time := 3599.5, [21].log_data[9].valid := 1, [21].log_data[10].min := 1.0, [21].log_data[10].max := 1.0, [21].log_data[10].total := 3599.5, [21].log_data[10].time := 3599.5, [21].log_data[10].valid := 1, [21].log_data[11].time := 3599.5, [21].log_data[11].valid := 1, [21].log_data[12].min := 1.0, [21].log_data[12].max := 1.0, [21].log_data[12].total := 3599.5, [21].log_data[12].time := 3599.5, [21].log_data[12].valid := 1, [21].log_data[13].min := 1.0, [21].log_data[13].max := 1.0, [21].log_data[13].total := 3599.5, [21].log_data[13].time := 3599.5, [21].log_data[13].valid := 1, [21].log_data[14].time := 3599.5, [21].log_data[14].valid := 1,
        [21].log_data[15].time := 3599.5, [21].log_data[15].valid := 1, [21].log_data[16].time := 3599.5, [21].log_data[16].valid := 1, [21].log_data[17].min := 1.0, [21].log_data[17].max := 1.0, [21].log_data[17].total := 3599.5, [21].log_data[17].time := 3599.5, [21].log_data[17].valid := 1, [21].log_data[18].time := 3599.5, [21].log_data[18].valid := 1, [21].log_data[19].time := 3599.5, [21].log_data[19].valid := 1, [21].log_data[20].time := 3599.5, [21].log_data[20].valid := 1, [21].log_data[21].min := 1.0, [21].log_data[21].max := 1.0, [21].log_data[21].total := 3599.5, [21].log_data[21].time := 3599.5, [21].log_data[21].valid := 1, [21].log_data[22].time := 3599.5, [21].log_data[22].valid := 1, [21].log_data[23].time := 3599.5, [21].log_data[23].valid := 1, [21].log_data[24].time := 3599.5, [21].log_data[24].valid := 1, [21].log_data[25].time := 3599.5, [21].log_data[25].valid := 1, [21].log_data[26].time := 3599.5, [21].log_data[26].valid := 1, [21].log_data[27].time := 3599.5, [21].log_data[27].valid := 1, [21].log_data[28].time := 3599.5, [21].log_data[28].valid := 1, [21].log_data[29].min := 1.0, [21].log_data[29].max := 1.0, [21].log_data[29].total := 3599.5, [21].log_data[29].time := 3599.5, [21].log_data[29].valid := 1, [21].log_data[30].min := 1.0, [21].log_data[30].max := 1.0, [21].log_data[30].total := 3599.5, [21].log_data[30].time := 3599.5, [21].log_data[30].valid := 1, [21].log_data[31].max := 1.0, [21].log_data[31].total := 1477.749, [21].log_data[31].time := 3599.5, [21].log_data[31].minminute := 6, [21].log_data[31].valid := 1, [21].log_data[32].max := 1.0, [21].log_data[32].total := 1629.7471, [21].log_data[32].time := 3599.5, [21].log_data[32].maxminute := 7, [21].log_data[32].valid := 1, [21].log_data[33].time := 3599.5, [21].log_data[33].valid := 1, [21].log_data[34].time := 3599.5, [21].log_data[34].valid := 1, [21].log_data[35].max := 1.0, [21].log_data[35].total := 1439.249,
        [21].log_data[35].time := 3599.5, [21].log_data[35].valid := 1, [21].log_data[36].max := 1.0, [21].log_data[36].total := 1629.998, [21].log_data[36].time := 3599.5, [21].log_data[36].maxminute := 2, [21].log_data[36].valid := 1, [21].log_data[37].max := 7.230523, [21].log_data[37].total := 3504.4326, [21].log_data[37].time := 3599.5, [21].log_data[37].maxminute := 9, [21].log_data[37].valid := 1, [21].log_data[38].time := 3599.5, [21].log_data[38].valid := 1, [21].log_data[39].min := 0.9950596, [21].log_data[39].max := 1.0227365, [21].log_data[39].total := 3609.4802, [21].log_data[39].time := 3599.5, [21].log_data[39].minminute := 47, [21].log_data[39].maxminute := 15, [21].log_data[39].valid := 1, [21].log_data[40].min := 7.5629425, [21].log_data[40].max := 7.5879498, [21].log_data[40].total := 27281.094, [21].log_data[40].time := 3599.5, [21].log_data[40].minminute := 25, [21].log_data[40].maxminute := 7, [21].log_data[40].valid := 1, [21].log_data[41].min := 0.039224852, [21].log_data[41].max := 0.06906128, [21].log_data[41].total := 174.52693, [21].log_data[41].time := 3599.5, [21].log_data[41].minminute := 9, [21].log_data[41].maxminute := 27, [21].log_data[41].valid := 1, [21].log_data[42].min := 2.2927027, [21].log_data[42].max := 2.2980025, [21].log_data[42].total := 8262.36, [21].log_data[42].time := 3599.5, [21].log_data[42].minminute := 23, [21].log_data[42].maxminute := 45, [21].log_data[42].valid := 1, [21].log_data[43].min := -0.27999878, [21].log_data[43].max := -0.26000214, [21].log_data[43].total := -935.8482, [21].log_data[43].time := 3599.5, [21].log_data[43].minminute := 17, [21].log_data[43].valid := 1, [21].log_data[44].min := -0.30000305, [21].log_data[44].max := -0.27999878, [21].log_data[44].total := -1044.0765, [21].log_data[44].time := 3599.5, [21].log_data[44].valid := 1, [21].log_data[45].time := 3599.5, [21].log_data[45].valid := 1, [21].log_data[46].time := 3599.5, [21].log_data[46].valid := 1, [21].log_data[47].time := 3599.5, [21].log_data[47].valid := 1, [21].log_data[48].min := 6.5810537,
        [21].log_data[48].max := 6.9223657, [21].log_data[48].total := 24213.94, [21].log_data[48].time := 3599.5, [21].log_data[48].minminute := 41, [21].log_data[48].maxminute := 13, [21].log_data[48].valid := 1, [21].log_data[49].min := 6.909816, [21].log_data[49].max := 9.553862, [21].log_data[49].total := 29291.77, [21].log_data[49].time := 3599.5, [21].log_data[49].minminute := 35, [21].log_data[49].maxminute := 9, [21].log_data[49].valid := 1, [21].log_data[50].min := 2.0224094, [21].log_data[50].max := 2.1300557, [21].log_data[50].total := 7513.9697, [21].log_data[50].time := 3599.5, [21].log_data[50].minminute := 10, [21].log_data[50].maxminute := 20, [21].log_data[50].valid := 1, [21].log_data[51].time := 3599.5, [21].log_data[51].valid := 1, [21].log_data[52].min := -2.840004, [21].log_data[52].max := 0.13999939, [21].log_data[52].total := -7599.141, [21].log_data[52].time := 3599.5, [21].log_data[52].minminute := 29, [21].log_data[52].maxminute := 38, [21].log_data[52].valid := 1, [21].log_data[53].min := -2.5, [21].log_data[53].max := 0.22000122, [21].log_data[53].total := -7043.792, [21].log_data[53].time := 3599.5, [21].log_data[53].minminute := 35, [21].log_data[53].maxminute := 2, [21].log_data[53].valid := 1, [21].log_data[54].max := 0.5285, [21].log_data[54].total := 1234.0566, [21].log_data[54].time := 3599.5, [21].log_data[54].minminute := 6, [21].log_data[54].maxminute := 39, [21].log_data[54].valid := 1, [21].log_data[55].max := 0.5295, [21].log_data[55].total := 1217.1123, [21].log_data[55].time := 3599.5, [21].log_data[55].maxminute := 54, [21].log_data[55].valid := 1, [21].log_data[56].min := 0.16020635, [21].log_data[56].max := 0.16067745, [21].log_data[56].total := 577.4519, [21].log_data[56].time := 3599.5, [21].log_data[56].minminute := 43, [21].log_data[56].maxminute := 4, [21].log_data[56].valid := 1, [21].log_data[57].min := 0.30232134, [21].log_data[57].max := 0.30420572, [21].log_data[57].total := 1092.689, [21].log_data[57].time := 3599.5, [21].log_data[57].minminute := 57, [21].log_data[57].maxminute := 5,
        [21].log_data[57].valid := 1, [21].log_data[58].time := 3599.5, [21].log_data[58].valid := 1, [21].log_data[59].time := 3599.5, [21].log_data[59].valid := 1, [21].log_data[60].valid := 1, [21].log_data[61].valid := 1, [21].log_data[62].valid := 1, [21].log_data[63].valid := 1, [21].log_data[64].valid := 1, [21].log_data[65].valid := 1, [21].log_data[66].valid := 1, [21].log_data[67].valid := 1, [21].log_data[68].valid := 1, [21].log_data[69].valid := 1, [21].log_data[70].valid := 1, [21].log_data[71].valid := 1, [21].log_data[72].valid := 1, [21].log_data[73].valid := 1, [21].log_data[74].valid := 1, [21].log_data[75].valid := 1, [21].log_data[76].valid := 1, [21].log_data[77].valid := 1, [21].log_data[78].valid := 1, [21].log_data[79].valid := 1, [21].log_data[80].valid := 1, [21].log_data[81].valid := 1, [21].log_data[82].valid := 1, [21].log_data[83].valid := 1, [21].log_data[84].valid := 1, [21].log_data[85].valid := 1, [21].log_data[86].valid := 1, [21].log_data[87].valid := 1, [21].log_data[88].valid := 1, [21].log_data[89].valid := 1, [21].log_data[90].valid := 1, [21].log_data[91].valid := 1, [21].log_data[92].valid := 1, [21].log_data[93].valid := 1, [21].log_data[94].valid := 1, [21].log_data[95].valid := 1, [21].log_data[96].valid := 1, [21].log_data[97].valid := 1, [21].log_data[98].valid := 1, [21].log_data[99].valid := 1, [21].log_data[100].valid := 1, [21].log_data[101].valid := 1, [21].log_data[102].valid := 1, [21].log_data[103].valid := 1, [21].log_data[104].valid := 1, [21].log_data[105].valid := 1, [21].log_data[106].valid := 1, [21].log_data[107].valid := 1, [21].log_data[108].valid := 1, [21].log_data[109].valid := 1, [21].log_data[110].valid := 1, [21].log_data[111].valid := 1, [21].log_data[112].valid := 1, [21].log_data[113].valid := 1, [21].log_data[114].valid := 1,
        [21].log_data[115].valid := 1, [21].log_data[116].valid := 1, [21].log_data[117].valid := 1, [21].log_data[118].valid := 1, [21].log_data[119].valid := 1, [21].log_data[120].valid := 1, [21].log_data[121].valid := 1, [21].log_data[122].valid := 1, [21].log_data[123].valid := 1, [21].log_data[124].valid := 1, [21].time.Year := 2023, [21].time.Month := 1, [21].time.Day := 14, [21].time.Minute := 59, [21].time.Second := 59, [22].log_data[0].min := 1.0, [22].log_data[0].max := 1.0, [22].log_data[0].total := 3600.0, [22].log_data[0].time := 3600.0, [22].log_data[0].valid := 1, [22].log_data[1].time := 3600.0, [22].log_data[1].valid := 1, [22].log_data[2].time := 3600.0, [22].log_data[2].valid := 1, [22].log_data[3].time := 3600.0, [22].log_data[3].valid := 1, [22].log_data[4].time := 3600.0, [22].log_data[4].valid := 1, [22].log_data[5].time := 3600.0, [22].log_data[5].valid := 1, [22].log_data[6].time := 3600.0, [22].log_data[6].valid := 1, [22].log_data[7].time := 3600.0, [22].log_data[7].valid := 1, [22].log_data[8].max := 1.0, [22].log_data[8].total := 3299.751, [22].log_data[8].time := 3600.0, [22].log_data[8].minminute := 54, [22].log_data[8].valid := 1, [22].log_data[9].max := 1.0, [22].log_data[9].total := 3299.751, [22].log_data[9].time := 3600.0, [22].log_data[9].minminute := 54, [22].log_data[9].valid := 1, [22].log_data[10].min := 1.0, [22].log_data[10].max := 1.0, [22].log_data[10].total := 3600.0, [22].log_data[10].time := 3600.0, [22].log_data[10].valid := 1, [22].log_data[11].time := 3600.0, [22].log_data[11].valid := 1, [22].log_data[12].min := 1.0, [22].log_data[12].max := 1.0, [22].log_data[12].total := 3600.0, [22].log_data[12].time := 3600.0, [22].log_data[12].valid := 1, [22].log_data[13].min := 1.0, [22].log_data[13].max := 1.0, [22].log_data[13].total := 3600.0, [22].log_data[13].time := 3600.0,
        [22].log_data[13].valid := 1, [22].log_data[14].time := 3600.0, [22].log_data[14].valid := 1, [22].log_data[15].time := 3600.0, [22].log_data[15].valid := 1, [22].log_data[16].time := 3600.0, [22].log_data[16].valid := 1, [22].log_data[17].min := 1.0, [22].log_data[17].max := 1.0, [22].log_data[17].total := 3600.0, [22].log_data[17].time := 3600.0, [22].log_data[17].valid := 1, [22].log_data[18].time := 3600.0, [22].log_data[18].valid := 1, [22].log_data[19].time := 3600.0, [22].log_data[19].valid := 1, [22].log_data[20].time := 3600.0, [22].log_data[20].valid := 1, [22].log_data[21].min := 1.0, [22].log_data[21].max := 1.0, [22].log_data[21].total := 3600.0, [22].log_data[21].time := 3600.0, [22].log_data[21].valid := 1, [22].log_data[22].time := 3600.0, [22].log_data[22].valid := 1, [22].log_data[23].time := 3600.0, [22].log_data[23].valid := 1, [22].log_data[24].time := 3600.0, [22].log_data[24].valid := 1, [22].log_data[25].time := 3600.0, [22].log_data[25].valid := 1, [22].log_data[26].time := 3600.0, [22].log_data[26].valid := 1, [22].log_data[27].time := 3600.0, [22].log_data[27].valid := 1, [22].log_data[28].time := 3600.0, [22].log_data[28].valid := 1, [22].log_data[29].min := 1.0, [22].log_data[29].max := 1.0, [22].log_data[29].total := 3600.0, [22].log_data[29].time := 3600.0, [22].log_data[29].valid := 1, [22].log_data[30].min := 1.0, [22].log_data[30].max := 1.0, [22].log_data[30].total := 3600.0, [22].log_data[30].time := 3600.0, [22].log_data[30].valid := 1, [22].log_data[31].max := 1.0, [22].log_data[31].total := 1629.498, [22].log_data[31].time := 3600.0, [22].log_data[31].valid := 1, [22].log_data[32].max := 1.0, [22].log_data[32].total := 1194.998, [22].log_data[32].time := 3600.0, [22].log_data[32].maxminute := 11, [22].log_data[32].valid := 1, [22].log_data[33].time := 3600.0, [22].log_data[33].valid := 1, [22].log_data[34].time := 3600.0, [22].log_data[34].valid := 1,
